  STRUCT
   STAT0 : ARRAY  [-32768 .. -30271 ] OF BYTE ;
  END_STRUCT ;
BEGIN
   STAT0[-32768] := B#16#0;
   STAT0[-32767] := B#16#0;
   STAT0[-32766] := B#16#0;
   STAT0[-32765] := B#16#0;
   STAT0[-32764] := B#16#0;
   STAT0[-32763] := B#16#1;
   STAT0[-32762] := B#16#0;
   STAT0[-32761] := B#16#0;
   STAT0[-32760] := B#16#0;
   STAT0[-32759] := B#16#1;
   STAT0[-32758] := B#16#0;
   STAT0[-32757] := B#16#1;
   STAT0[-32756] := B#16#0;
   STAT0[-32755] := B#16#1;
   STAT0[-32754] := B#16#0;
   STAT0[-32753] := B#16#1;
   STAT0[-32752] := B#16#0;
   STAT0[-32751] := B#16#1;
   STAT0[-32750] := B#16#0;
   STAT0[-32749] := B#16#1;
   STAT0[-32748] := B#16#0;
   STAT0[-32747] := B#16#1;
   STAT0[-32746] := B#16#0;
   STAT0[-32745] := B#16#1;
   STAT0[-32744] := B#16#0;
   STAT0[-32743] := B#16#1;
   STAT0[-32742] := B#16#0;
   STAT0[-32741] := B#16#1;
   STAT0[-32740] := B#16#0;
   STAT0[-32739] := B#16#1;
   STAT0[-32738] := B#16#0;
   STAT0[-32737] := B#16#0;
   STAT0[-32736] := B#16#0;
   STAT0[-32735] := B#16#0;
   STAT0[-32734] := B#16#0;
   STAT0[-32733] := B#16#0;
   STAT0[-32732] := B#16#0;
   STAT0[-32731] := B#16#0;
   STAT0[-32730] := B#16#0;
   STAT0[-32729] := B#16#0;
   STAT0[-32728] := B#16#0;
   STAT0[-32727] := B#16#0;
   STAT0[-32726] := B#16#0;
   STAT0[-32725] := B#16#0;
   STAT0[-32724] := B#16#0;
   STAT0[-32723] := B#16#0;
   STAT0[-32722] := B#16#0;
   STAT0[-32721] := B#16#0;
   STAT0[-32720] := B#16#0;
   STAT0[-32719] := B#16#0;
   STAT0[-32718] := B#16#0;
   STAT0[-32717] := B#16#0;
   STAT0[-32716] := B#16#0;
   STAT0[-32715] := B#16#0;
   STAT0[-32714] := B#16#0;
   STAT0[-32713] := B#16#0;
   STAT0[-32712] := B#16#0;
   STAT0[-32711] := B#16#0;
   STAT0[-32710] := B#16#0;
   STAT0[-32709] := B#16#0;
   STAT0[-32708] := B#16#0;
   STAT0[-32707] := B#16#0;
   STAT0[-32706] := B#16#0;
   STAT0[-32705] := B#16#0;
   STAT0[-32704] := B#16#0;
   STAT0[-32703] := B#16#0;
   STAT0[-32702] := B#16#0;
   STAT0[-32701] := B#16#0;
   STAT0[-32700] := B#16#0;
   STAT0[-32699] := B#16#0;
   STAT0[-32698] := B#16#0;
   STAT0[-32697] := B#16#0;
   STAT0[-32696] := B#16#0;
   STAT0[-32695] := B#16#0;
   STAT0[-32694] := B#16#0;
   STAT0[-32693] := B#16#0;
   STAT0[-32692] := B#16#0;
   STAT0[-32691] := B#16#0;
   STAT0[-32690] := B#16#0;
   STAT0[-32689] := B#16#0;
   STAT0[-32688] := B#16#0;
   STAT0[-32687] := B#16#0;
   STAT0[-32686] := B#16#0;
   STAT0[-32685] := B#16#0;
   STAT0[-32684] := B#16#0;
   STAT0[-32683] := B#16#0;
   STAT0[-32682] := B#16#0;
   STAT0[-32681] := B#16#0;
   STAT0[-32680] := B#16#0;
   STAT0[-32679] := B#16#0;
   STAT0[-32678] := B#16#0;
   STAT0[-32677] := B#16#0;
   STAT0[-32676] := B#16#0;
   STAT0[-32675] := B#16#0;
   STAT0[-32674] := B#16#0;
   STAT0[-32673] := B#16#0;
   STAT0[-32672] := B#16#0;
   STAT0[-32671] := B#16#0;
   STAT0[-32670] := B#16#0;
   STAT0[-32669] := B#16#0;
   STAT0[-32668] := B#16#0;
   STAT0[-32667] := B#16#0;
   STAT0[-32666] := B#16#0;
   STAT0[-32665] := B#16#0;
   STAT0[-32664] := B#16#0;
   STAT0[-32663] := B#16#0;
   STAT0[-32662] := B#16#0;
   STAT0[-32661] := B#16#0;
   STAT0[-32660] := B#16#0;
   STAT0[-32659] := B#16#0;
   STAT0[-32658] := B#16#0;
   STAT0[-32657] := B#16#0;
   STAT0[-32656] := B#16#0;
   STAT0[-32655] := B#16#0;
   STAT0[-32654] := B#16#0;
   STAT0[-32653] := B#16#0;
   STAT0[-32652] := B#16#0;
   STAT0[-32651] := B#16#0;
   STAT0[-32650] := B#16#0;
   STAT0[-32649] := B#16#0;
   STAT0[-32648] := B#16#0;
   STAT0[-32647] := B#16#0;
   STAT0[-32646] := B#16#0;
   STAT0[-32645] := B#16#0;
   STAT0[-32644] := B#16#0;
   STAT0[-32643] := B#16#0;
   STAT0[-32642] := B#16#0;
   STAT0[-32641] := B#16#0;
   STAT0[-32640] := B#16#0;
   STAT0[-32639] := B#16#0;
   STAT0[-32638] := B#16#0;
   STAT0[-32637] := B#16#0;
   STAT0[-32636] := B#16#0;
   STAT0[-32635] := B#16#0;
   STAT0[-32634] := B#16#0;
   STAT0[-32633] := B#16#0;
   STAT0[-32632] := B#16#0;
   STAT0[-32631] := B#16#0;
   STAT0[-32630] := B#16#0;
   STAT0[-32629] := B#16#0;
   STAT0[-32628] := B#16#0;
   STAT0[-32627] := B#16#0;
   STAT0[-32626] := B#16#0;
   STAT0[-32625] := B#16#0;
   STAT0[-32624] := B#16#0;
   STAT0[-32623] := B#16#0;
   STAT0[-32622] := B#16#0;
   STAT0[-32621] := B#16#0;
   STAT0[-32620] := B#16#0;
   STAT0[-32619] := B#16#0;
   STAT0[-32618] := B#16#0;
   STAT0[-32617] := B#16#0;
   STAT0[-32616] := B#16#0;
   STAT0[-32615] := B#16#0;
   STAT0[-32614] := B#16#0;
   STAT0[-32613] := B#16#0;
   STAT0[-32612] := B#16#0;
   STAT0[-32611] := B#16#0;
   STAT0[-32610] := B#16#0;
   STAT0[-32609] := B#16#0;
   STAT0[-32608] := B#16#0;
   STAT0[-32607] := B#16#0;
   STAT0[-32606] := B#16#0;
   STAT0[-32605] := B#16#0;
   STAT0[-32604] := B#16#0;
   STAT0[-32603] := B#16#0;
   STAT0[-32602] := B#16#0;
   STAT0[-32601] := B#16#0;
   STAT0[-32600] := B#16#0;
   STAT0[-32599] := B#16#0;
   STAT0[-32598] := B#16#0;
   STAT0[-32597] := B#16#0;
   STAT0[-32596] := B#16#0;
   STAT0[-32595] := B#16#0;
   STAT0[-32594] := B#16#0;
   STAT0[-32593] := B#16#0;
   STAT0[-32592] := B#16#0;
   STAT0[-32591] := B#16#0;
   STAT0[-32590] := B#16#0;
   STAT0[-32589] := B#16#0;
   STAT0[-32588] := B#16#0;
   STAT0[-32587] := B#16#0;
   STAT0[-32586] := B#16#0;
   STAT0[-32585] := B#16#0;
   STAT0[-32584] := B#16#0;
   STAT0[-32583] := B#16#0;
   STAT0[-32582] := B#16#0;
   STAT0[-32581] := B#16#0;
   STAT0[-32580] := B#16#0;
   STAT0[-32579] := B#16#0;
   STAT0[-32578] := B#16#0;
   STAT0[-32577] := B#16#0;
   STAT0[-32576] := B#16#0;
   STAT0[-32575] := B#16#0;
   STAT0[-32574] := B#16#0;
   STAT0[-32573] := B#16#0;
   STAT0[-32572] := B#16#0;
   STAT0[-32571] := B#16#0;
   STAT0[-32570] := B#16#0;
   STAT0[-32569] := B#16#0;
   STAT0[-32568] := B#16#0;
   STAT0[-32567] := B#16#0;
   STAT0[-32566] := B#16#0;
   STAT0[-32565] := B#16#0;
   STAT0[-32564] := B#16#0;
   STAT0[-32563] := B#16#0;
   STAT0[-32562] := B#16#0;
   STAT0[-32561] := B#16#0;
   STAT0[-32560] := B#16#0;
   STAT0[-32559] := B#16#0;
   STAT0[-32558] := B#16#0;
   STAT0[-32557] := B#16#0;
   STAT0[-32556] := B#16#0;
   STAT0[-32555] := B#16#0;
   STAT0[-32554] := B#16#0;
   STAT0[-32553] := B#16#0;
   STAT0[-32552] := B#16#0;
   STAT0[-32551] := B#16#0;
   STAT0[-32550] := B#16#0;
   STAT0[-32549] := B#16#0;
   STAT0[-32548] := B#16#0;
   STAT0[-32547] := B#16#0;
   STAT0[-32546] := B#16#0;
   STAT0[-32545] := B#16#0;
   STAT0[-32544] := B#16#0;
   STAT0[-32543] := B#16#0;
   STAT0[-32542] := B#16#0;
   STAT0[-32541] := B#16#0;
   STAT0[-32540] := B#16#0;
   STAT0[-32539] := B#16#0;
   STAT0[-32538] := B#16#0;
   STAT0[-32537] := B#16#0;
   STAT0[-32536] := B#16#0;
   STAT0[-32535] := B#16#0;
   STAT0[-32534] := B#16#0;
   STAT0[-32533] := B#16#0;
   STAT0[-32532] := B#16#0;
   STAT0[-32531] := B#16#0;
   STAT0[-32530] := B#16#0;
   STAT0[-32529] := B#16#0;
   STAT0[-32528] := B#16#0;
   STAT0[-32527] := B#16#0;
   STAT0[-32526] := B#16#0;
   STAT0[-32525] := B#16#0;
   STAT0[-32524] := B#16#0;
   STAT0[-32523] := B#16#0;
   STAT0[-32522] := B#16#0;
   STAT0[-32521] := B#16#0;
   STAT0[-32520] := B#16#0;
   STAT0[-32519] := B#16#0;
   STAT0[-32518] := B#16#0;
   STAT0[-32517] := B#16#0;
   STAT0[-32516] := B#16#0;
   STAT0[-32515] := B#16#0;
   STAT0[-32514] := B#16#0;
   STAT0[-32513] := B#16#0;
   STAT0[-32512] := B#16#0;
   STAT0[-32511] := B#16#0;
   STAT0[-32510] := B#16#0;
   STAT0[-32509] := B#16#0;
   STAT0[-32508] := B#16#0;
   STAT0[-32507] := B#16#0;
   STAT0[-32506] := B#16#0;
   STAT0[-32505] := B#16#0;
   STAT0[-32504] := B#16#0;
   STAT0[-32503] := B#16#0;
   STAT0[-32502] := B#16#0;
   STAT0[-32501] := B#16#0;
   STAT0[-32500] := B#16#0;
   STAT0[-32499] := B#16#0;
   STAT0[-32498] := B#16#0;
   STAT0[-32497] := B#16#0;
   STAT0[-32496] := B#16#0;
   STAT0[-32495] := B#16#0;
   STAT0[-32494] := B#16#0;
   STAT0[-32493] := B#16#0;
   STAT0[-32492] := B#16#0;
   STAT0[-32491] := B#16#0;
   STAT0[-32490] := B#16#0;
   STAT0[-32489] := B#16#0;
   STAT0[-32488] := B#16#0;
   STAT0[-32487] := B#16#0;
   STAT0[-32486] := B#16#0;
   STAT0[-32485] := B#16#0;
   STAT0[-32484] := B#16#0;
   STAT0[-32483] := B#16#0;
   STAT0[-32482] := B#16#0;
   STAT0[-32481] := B#16#0;
   STAT0[-32480] := B#16#0;
   STAT0[-32479] := B#16#0;
   STAT0[-32478] := B#16#0;
   STAT0[-32477] := B#16#0;
   STAT0[-32476] := B#16#0;
   STAT0[-32475] := B#16#0;
   STAT0[-32474] := B#16#0;
   STAT0[-32473] := B#16#0;
   STAT0[-32472] := B#16#0;
   STAT0[-32471] := B#16#0;
   STAT0[-32470] := B#16#0;
   STAT0[-32469] := B#16#0;
   STAT0[-32468] := B#16#0;
   STAT0[-32467] := B#16#0;
   STAT0[-32466] := B#16#0;
   STAT0[-32465] := B#16#0;
   STAT0[-32464] := B#16#0;
   STAT0[-32463] := B#16#0;
   STAT0[-32462] := B#16#0;
   STAT0[-32461] := B#16#0;
   STAT0[-32460] := B#16#0;
   STAT0[-32459] := B#16#0;
   STAT0[-32458] := B#16#0;
   STAT0[-32457] := B#16#0;
   STAT0[-32456] := B#16#0;
   STAT0[-32455] := B#16#0;
   STAT0[-32454] := B#16#0;
   STAT0[-32453] := B#16#0;
   STAT0[-32452] := B#16#0;
   STAT0[-32451] := B#16#0;
   STAT0[-32450] := B#16#0;
   STAT0[-32449] := B#16#0;
   STAT0[-32448] := B#16#0;
   STAT0[-32447] := B#16#0;
   STAT0[-32446] := B#16#0;
   STAT0[-32445] := B#16#0;
   STAT0[-32444] := B#16#0;
   STAT0[-32443] := B#16#0;
   STAT0[-32442] := B#16#0;
   STAT0[-32441] := B#16#0;
   STAT0[-32440] := B#16#0;
   STAT0[-32439] := B#16#0;
   STAT0[-32438] := B#16#0;
   STAT0[-32437] := B#16#0;
   STAT0[-32436] := B#16#0;
   STAT0[-32435] := B#16#0;
   STAT0[-32434] := B#16#0;
   STAT0[-32433] := B#16#0;
   STAT0[-32432] := B#16#0;
   STAT0[-32431] := B#16#0;
   STAT0[-32430] := B#16#0;
   STAT0[-32429] := B#16#0;
   STAT0[-32428] := B#16#0;
   STAT0[-32427] := B#16#0;
   STAT0[-32426] := B#16#0;
   STAT0[-32425] := B#16#0;
   STAT0[-32424] := B#16#0;
   STAT0[-32423] := B#16#0;
   STAT0[-32422] := B#16#0;
   STAT0[-32421] := B#16#0;
   STAT0[-32420] := B#16#0;
   STAT0[-32419] := B#16#0;
   STAT0[-32418] := B#16#0;
   STAT0[-32417] := B#16#0;
   STAT0[-32416] := B#16#0;
   STAT0[-32415] := B#16#0;
   STAT0[-32414] := B#16#0;
   STAT0[-32413] := B#16#0;
   STAT0[-32412] := B#16#0;
   STAT0[-32411] := B#16#0;
   STAT0[-32410] := B#16#0;
   STAT0[-32409] := B#16#0;
   STAT0[-32408] := B#16#0;
   STAT0[-32407] := B#16#0;
   STAT0[-32406] := B#16#0;
   STAT0[-32405] := B#16#0;
   STAT0[-32404] := B#16#0;
   STAT0[-32403] := B#16#0;
   STAT0[-32402] := B#16#0;
   STAT0[-32401] := B#16#0;
   STAT0[-32400] := B#16#0;
   STAT0[-32399] := B#16#0;
   STAT0[-32398] := B#16#0;
   STAT0[-32397] := B#16#0;
   STAT0[-32396] := B#16#0;
   STAT0[-32395] := B#16#0;
   STAT0[-32394] := B#16#0;
   STAT0[-32393] := B#16#0;
   STAT0[-32392] := B#16#0;
   STAT0[-32391] := B#16#0;
   STAT0[-32390] := B#16#0;
   STAT0[-32389] := B#16#0;
   STAT0[-32388] := B#16#0;
   STAT0[-32387] := B#16#0;
   STAT0[-32386] := B#16#0;
   STAT0[-32385] := B#16#0;
   STAT0[-32384] := B#16#0;
   STAT0[-32383] := B#16#0;
   STAT0[-32382] := B#16#0;
   STAT0[-32381] := B#16#0;
   STAT0[-32380] := B#16#0;
   STAT0[-32379] := B#16#0;
   STAT0[-32378] := B#16#0;
   STAT0[-32377] := B#16#0;
   STAT0[-32376] := B#16#0;
   STAT0[-32375] := B#16#0;
   STAT0[-32374] := B#16#0;
   STAT0[-32373] := B#16#0;
   STAT0[-32372] := B#16#0;
   STAT0[-32371] := B#16#0;
   STAT0[-32370] := B#16#0;
   STAT0[-32369] := B#16#0;
   STAT0[-32368] := B#16#0;
   STAT0[-32367] := B#16#0;
   STAT0[-32366] := B#16#0;
   STAT0[-32365] := B#16#0;
   STAT0[-32364] := B#16#0;
   STAT0[-32363] := B#16#0;
   STAT0[-32362] := B#16#0;
   STAT0[-32361] := B#16#0;
   STAT0[-32360] := B#16#0;
   STAT0[-32359] := B#16#0;
   STAT0[-32358] := B#16#0;
   STAT0[-32357] := B#16#0;
   STAT0[-32356] := B#16#0;
   STAT0[-32355] := B#16#0;
   STAT0[-32354] := B#16#0;
   STAT0[-32353] := B#16#0;
   STAT0[-32352] := B#16#0;
   STAT0[-32351] := B#16#0;
   STAT0[-32350] := B#16#0;
   STAT0[-32349] := B#16#0;
   STAT0[-32348] := B#16#0;
   STAT0[-32347] := B#16#0;
   STAT0[-32346] := B#16#0;
   STAT0[-32345] := B#16#0;
   STAT0[-32344] := B#16#0;
   STAT0[-32343] := B#16#0;
   STAT0[-32342] := B#16#0;
   STAT0[-32341] := B#16#0;
   STAT0[-32340] := B#16#0;
   STAT0[-32339] := B#16#0;
   STAT0[-32338] := B#16#0;
   STAT0[-32337] := B#16#0;
   STAT0[-32336] := B#16#0;
   STAT0[-32335] := B#16#0;
   STAT0[-32334] := B#16#0;
   STAT0[-32333] := B#16#0;
   STAT0[-32332] := B#16#0;
   STAT0[-32331] := B#16#0;
   STAT0[-32330] := B#16#0;
   STAT0[-32329] := B#16#0;
   STAT0[-32328] := B#16#0;
   STAT0[-32327] := B#16#0;
   STAT0[-32326] := B#16#0;
   STAT0[-32325] := B#16#0;
   STAT0[-32324] := B#16#0;
   STAT0[-32323] := B#16#0;
   STAT0[-32322] := B#16#0;
   STAT0[-32321] := B#16#0;
   STAT0[-32320] := B#16#0;
   STAT0[-32319] := B#16#0;
   STAT0[-32318] := B#16#0;
   STAT0[-32317] := B#16#0;
   STAT0[-32316] := B#16#0;
   STAT0[-32315] := B#16#0;
   STAT0[-32314] := B#16#0;
   STAT0[-32313] := B#16#0;
   STAT0[-32312] := B#16#0;
   STAT0[-32311] := B#16#0;
   STAT0[-32310] := B#16#0;
   STAT0[-32309] := B#16#0;
   STAT0[-32308] := B#16#0;
   STAT0[-32307] := B#16#0;
   STAT0[-32306] := B#16#0;
   STAT0[-32305] := B#16#0;
   STAT0[-32304] := B#16#0;
   STAT0[-32303] := B#16#0;
   STAT0[-32302] := B#16#0;
   STAT0[-32301] := B#16#0;
   STAT0[-32300] := B#16#0;
   STAT0[-32299] := B#16#0;
   STAT0[-32298] := B#16#0;
   STAT0[-32297] := B#16#0;
   STAT0[-32296] := B#16#0;
   STAT0[-32295] := B#16#0;
   STAT0[-32294] := B#16#0;
   STAT0[-32293] := B#16#0;
   STAT0[-32292] := B#16#0;
   STAT0[-32291] := B#16#0;
   STAT0[-32290] := B#16#0;
   STAT0[-32289] := B#16#0;
   STAT0[-32288] := B#16#0;
   STAT0[-32287] := B#16#0;
   STAT0[-32286] := B#16#0;
   STAT0[-32285] := B#16#0;
   STAT0[-32284] := B#16#0;
   STAT0[-32283] := B#16#0;
   STAT0[-32282] := B#16#0;
   STAT0[-32281] := B#16#0;
   STAT0[-32280] := B#16#0;
   STAT0[-32279] := B#16#0;
   STAT0[-32278] := B#16#0;
   STAT0[-32277] := B#16#0;
   STAT0[-32276] := B#16#0;
   STAT0[-32275] := B#16#0;
   STAT0[-32274] := B#16#0;
   STAT0[-32273] := B#16#0;
   STAT0[-32272] := B#16#0;
   STAT0[-32271] := B#16#0;
   STAT0[-32270] := B#16#0;
   STAT0[-32269] := B#16#0;
   STAT0[-32268] := B#16#0;
   STAT0[-32267] := B#16#0;
   STAT0[-32266] := B#16#0;
   STAT0[-32265] := B#16#0;
   STAT0[-32264] := B#16#0;
   STAT0[-32263] := B#16#0;
   STAT0[-32262] := B#16#0;
   STAT0[-32261] := B#16#0;
   STAT0[-32260] := B#16#0;
   STAT0[-32259] := B#16#0;
   STAT0[-32258] := B#16#0;
   STAT0[-32257] := B#16#0;
   STAT0[-32256] := B#16#0;
   STAT0[-32255] := B#16#0;
   STAT0[-32254] := B#16#0;
   STAT0[-32253] := B#16#0;
   STAT0[-32252] := B#16#0;
   STAT0[-32251] := B#16#0;
   STAT0[-32250] := B#16#0;
   STAT0[-32249] := B#16#0;
   STAT0[-32248] := B#16#0;
   STAT0[-32247] := B#16#0;
   STAT0[-32246] := B#16#0;
   STAT0[-32245] := B#16#0;
   STAT0[-32244] := B#16#0;
   STAT0[-32243] := B#16#0;
   STAT0[-32242] := B#16#0;
   STAT0[-32241] := B#16#0;
   STAT0[-32240] := B#16#0;
   STAT0[-32239] := B#16#0;
   STAT0[-32238] := B#16#0;
   STAT0[-32237] := B#16#0;
   STAT0[-32236] := B#16#0;
   STAT0[-32235] := B#16#0;
   STAT0[-32234] := B#16#0;
   STAT0[-32233] := B#16#0;
   STAT0[-32232] := B#16#0;
   STAT0[-32231] := B#16#0;
   STAT0[-32230] := B#16#0;
   STAT0[-32229] := B#16#0;
   STAT0[-32228] := B#16#0;
   STAT0[-32227] := B#16#0;
   STAT0[-32226] := B#16#0;
   STAT0[-32225] := B#16#0;
   STAT0[-32224] := B#16#0;
   STAT0[-32223] := B#16#0;
   STAT0[-32222] := B#16#0;
   STAT0[-32221] := B#16#0;
   STAT0[-32220] := B#16#0;
   STAT0[-32219] := B#16#0;
   STAT0[-32218] := B#16#0;
   STAT0[-32217] := B#16#0;
   STAT0[-32216] := B#16#0;
   STAT0[-32215] := B#16#0;
   STAT0[-32214] := B#16#0;
   STAT0[-32213] := B#16#0;
   STAT0[-32212] := B#16#0;
   STAT0[-32211] := B#16#0;
   STAT0[-32210] := B#16#0;
   STAT0[-32209] := B#16#0;
   STAT0[-32208] := B#16#0;
   STAT0[-32207] := B#16#0;
   STAT0[-32206] := B#16#0;
   STAT0[-32205] := B#16#0;
   STAT0[-32204] := B#16#0;
   STAT0[-32203] := B#16#0;
   STAT0[-32202] := B#16#0;
   STAT0[-32201] := B#16#0;
   STAT0[-32200] := B#16#0;
   STAT0[-32199] := B#16#0;
   STAT0[-32198] := B#16#0;
   STAT0[-32197] := B#16#0;
   STAT0[-32196] := B#16#0;
   STAT0[-32195] := B#16#0;
   STAT0[-32194] := B#16#0;
   STAT0[-32193] := B#16#0;
   STAT0[-32192] := B#16#0;
   STAT0[-32191] := B#16#0;
   STAT0[-32190] := B#16#0;
   STAT0[-32189] := B#16#0;
   STAT0[-32188] := B#16#0;
   STAT0[-32187] := B#16#0;
   STAT0[-32186] := B#16#0;
   STAT0[-32185] := B#16#0;
   STAT0[-32184] := B#16#0;
   STAT0[-32183] := B#16#0;
   STAT0[-32182] := B#16#0;
   STAT0[-32181] := B#16#0;
   STAT0[-32180] := B#16#0;
   STAT0[-32179] := B#16#0;
   STAT0[-32178] := B#16#0;
   STAT0[-32177] := B#16#0;
   STAT0[-32176] := B#16#0;
   STAT0[-32175] := B#16#0;
   STAT0[-32174] := B#16#0;
   STAT0[-32173] := B#16#0;
   STAT0[-32172] := B#16#0;
   STAT0[-32171] := B#16#0;
   STAT0[-32170] := B#16#0;
   STAT0[-32169] := B#16#0;
   STAT0[-32168] := B#16#0;
   STAT0[-32167] := B#16#0;
   STAT0[-32166] := B#16#0;
   STAT0[-32165] := B#16#0;
   STAT0[-32164] := B#16#0;
   STAT0[-32163] := B#16#0;
   STAT0[-32162] := B#16#0;
   STAT0[-32161] := B#16#0;
   STAT0[-32160] := B#16#0;
   STAT0[-32159] := B#16#0;
   STAT0[-32158] := B#16#0;
   STAT0[-32157] := B#16#0;
   STAT0[-32156] := B#16#0;
   STAT0[-32155] := B#16#0;
   STAT0[-32154] := B#16#0;
   STAT0[-32153] := B#16#0;
   STAT0[-32152] := B#16#0;
   STAT0[-32151] := B#16#0;
   STAT0[-32150] := B#16#0;
   STAT0[-32149] := B#16#0;
   STAT0[-32148] := B#16#0;
   STAT0[-32147] := B#16#0;
   STAT0[-32146] := B#16#0;
   STAT0[-32145] := B#16#0;
   STAT0[-32144] := B#16#0;
   STAT0[-32143] := B#16#0;
   STAT0[-32142] := B#16#0;
   STAT0[-32141] := B#16#0;
   STAT0[-32140] := B#16#0;
   STAT0[-32139] := B#16#0;
   STAT0[-32138] := B#16#0;
   STAT0[-32137] := B#16#0;
   STAT0[-32136] := B#16#0;
   STAT0[-32135] := B#16#0;
   STAT0[-32134] := B#16#0;
   STAT0[-32133] := B#16#0;
   STAT0[-32132] := B#16#0;
   STAT0[-32131] := B#16#0;
   STAT0[-32130] := B#16#0;
   STAT0[-32129] := B#16#0;
   STAT0[-32128] := B#16#0;
   STAT0[-32127] := B#16#0;
   STAT0[-32126] := B#16#0;
   STAT0[-32125] := B#16#0;
   STAT0[-32124] := B#16#0;
   STAT0[-32123] := B#16#0;
   STAT0[-32122] := B#16#0;
   STAT0[-32121] := B#16#0;
   STAT0[-32120] := B#16#0;
   STAT0[-32119] := B#16#0;
   STAT0[-32118] := B#16#0;
   STAT0[-32117] := B#16#0;
   STAT0[-32116] := B#16#0;
   STAT0[-32115] := B#16#0;
   STAT0[-32114] := B#16#0;
   STAT0[-32113] := B#16#0;
   STAT0[-32112] := B#16#0;
   STAT0[-32111] := B#16#0;
   STAT0[-32110] := B#16#0;
   STAT0[-32109] := B#16#0;
   STAT0[-32108] := B#16#0;
   STAT0[-32107] := B#16#0;
   STAT0[-32106] := B#16#0;
   STAT0[-32105] := B#16#0;
   STAT0[-32104] := B#16#0;
   STAT0[-32103] := B#16#0;
   STAT0[-32102] := B#16#0;
   STAT0[-32101] := B#16#0;
   STAT0[-32100] := B#16#0;
   STAT0[-32099] := B#16#0;
   STAT0[-32098] := B#16#0;
   STAT0[-32097] := B#16#0;
   STAT0[-32096] := B#16#0;
   STAT0[-32095] := B#16#0;
   STAT0[-32094] := B#16#0;
   STAT0[-32093] := B#16#0;
   STAT0[-32092] := B#16#0;
   STAT0[-32091] := B#16#0;
   STAT0[-32090] := B#16#0;
   STAT0[-32089] := B#16#0;
   STAT0[-32088] := B#16#0;
   STAT0[-32087] := B#16#0;
   STAT0[-32086] := B#16#0;
   STAT0[-32085] := B#16#0;
   STAT0[-32084] := B#16#0;
   STAT0[-32083] := B#16#0;
   STAT0[-32082] := B#16#0;
   STAT0[-32081] := B#16#0;
   STAT0[-32080] := B#16#0;
   STAT0[-32079] := B#16#0;
   STAT0[-32078] := B#16#0;
   STAT0[-32077] := B#16#0;
   STAT0[-32076] := B#16#0;
   STAT0[-32075] := B#16#0;
   STAT0[-32074] := B#16#0;
   STAT0[-32073] := B#16#0;
   STAT0[-32072] := B#16#0;
   STAT0[-32071] := B#16#0;
   STAT0[-32070] := B#16#0;
   STAT0[-32069] := B#16#0;
   STAT0[-32068] := B#16#0;
   STAT0[-32067] := B#16#0;
   STAT0[-32066] := B#16#0;
   STAT0[-32065] := B#16#0;
   STAT0[-32064] := B#16#0;
   STAT0[-32063] := B#16#0;
   STAT0[-32062] := B#16#0;
   STAT0[-32061] := B#16#0;
   STAT0[-32060] := B#16#0;
   STAT0[-32059] := B#16#0;
   STAT0[-32058] := B#16#0;
   STAT0[-32057] := B#16#0;
   STAT0[-32056] := B#16#0;
   STAT0[-32055] := B#16#0;
   STAT0[-32054] := B#16#0;
   STAT0[-32053] := B#16#0;
   STAT0[-32052] := B#16#0;
   STAT0[-32051] := B#16#0;
   STAT0[-32050] := B#16#0;
   STAT0[-32049] := B#16#0;
   STAT0[-32048] := B#16#0;
   STAT0[-32047] := B#16#0;
   STAT0[-32046] := B#16#0;
   STAT0[-32045] := B#16#0;
   STAT0[-32044] := B#16#0;
   STAT0[-32043] := B#16#0;
   STAT0[-32042] := B#16#0;
   STAT0[-32041] := B#16#0;
   STAT0[-32040] := B#16#0;
   STAT0[-32039] := B#16#0;
   STAT0[-32038] := B#16#0;
   STAT0[-32037] := B#16#0;
   STAT0[-32036] := B#16#0;
   STAT0[-32035] := B#16#0;
   STAT0[-32034] := B#16#0;
   STAT0[-32033] := B#16#0;
   STAT0[-32032] := B#16#0;
   STAT0[-32031] := B#16#0;
   STAT0[-32030] := B#16#0;
   STAT0[-32029] := B#16#0;
   STAT0[-32028] := B#16#0;
   STAT0[-32027] := B#16#0;
   STAT0[-32026] := B#16#0;
   STAT0[-32025] := B#16#0;
   STAT0[-32024] := B#16#0;
   STAT0[-32023] := B#16#0;
   STAT0[-32022] := B#16#0;
   STAT0[-32021] := B#16#0;
   STAT0[-32020] := B#16#0;
   STAT0[-32019] := B#16#0;
   STAT0[-32018] := B#16#0;
   STAT0[-32017] := B#16#0;
   STAT0[-32016] := B#16#0;
   STAT0[-32015] := B#16#0;
   STAT0[-32014] := B#16#0;
   STAT0[-32013] := B#16#0;
   STAT0[-32012] := B#16#0;
   STAT0[-32011] := B#16#0;
   STAT0[-32010] := B#16#0;
   STAT0[-32009] := B#16#0;
   STAT0[-32008] := B#16#0;
   STAT0[-32007] := B#16#0;
   STAT0[-32006] := B#16#0;
   STAT0[-32005] := B#16#0;
   STAT0[-32004] := B#16#0;
   STAT0[-32003] := B#16#0;
   STAT0[-32002] := B#16#0;
   STAT0[-32001] := B#16#0;
   STAT0[-32000] := B#16#0;
   STAT0[-31999] := B#16#0;
   STAT0[-31998] := B#16#0;
   STAT0[-31997] := B#16#0;
   STAT0[-31996] := B#16#0;
   STAT0[-31995] := B#16#0;
   STAT0[-31994] := B#16#0;
   STAT0[-31993] := B#16#0;
   STAT0[-31992] := B#16#0;
   STAT0[-31991] := B#16#0;
   STAT0[-31990] := B#16#0;
   STAT0[-31989] := B#16#0;
   STAT0[-31988] := B#16#0;
   STAT0[-31987] := B#16#0;
   STAT0[-31986] := B#16#0;
   STAT0[-31985] := B#16#0;
   STAT0[-31984] := B#16#0;
   STAT0[-31983] := B#16#0;
   STAT0[-31982] := B#16#0;
   STAT0[-31981] := B#16#0;
   STAT0[-31980] := B#16#0;
   STAT0[-31979] := B#16#0;
   STAT0[-31978] := B#16#0;
   STAT0[-31977] := B#16#0;
   STAT0[-31976] := B#16#0;
   STAT0[-31975] := B#16#0;
   STAT0[-31974] := B#16#0;
   STAT0[-31973] := B#16#0;
   STAT0[-31972] := B#16#0;
   STAT0[-31971] := B#16#0;
   STAT0[-31970] := B#16#0;
   STAT0[-31969] := B#16#0;
   STAT0[-31968] := B#16#0;
   STAT0[-31967] := B#16#0;
   STAT0[-31966] := B#16#0;
   STAT0[-31965] := B#16#0;
   STAT0[-31964] := B#16#0;
   STAT0[-31963] := B#16#0;
   STAT0[-31962] := B#16#0;
   STAT0[-31961] := B#16#0;
   STAT0[-31960] := B#16#0;
   STAT0[-31959] := B#16#0;
   STAT0[-31958] := B#16#0;
   STAT0[-31957] := B#16#0;
   STAT0[-31956] := B#16#0;
   STAT0[-31955] := B#16#0;
   STAT0[-31954] := B#16#0;
   STAT0[-31953] := B#16#0;
   STAT0[-31952] := B#16#0;
   STAT0[-31951] := B#16#0;
   STAT0[-31950] := B#16#0;
   STAT0[-31949] := B#16#0;
   STAT0[-31948] := B#16#0;
   STAT0[-31947] := B#16#0;
   STAT0[-31946] := B#16#0;
   STAT0[-31945] := B#16#0;
   STAT0[-31944] := B#16#0;
   STAT0[-31943] := B#16#0;
   STAT0[-31942] := B#16#0;
   STAT0[-31941] := B#16#0;
   STAT0[-31940] := B#16#0;
   STAT0[-31939] := B#16#0;
   STAT0[-31938] := B#16#0;
   STAT0[-31937] := B#16#0;
   STAT0[-31936] := B#16#0;
   STAT0[-31935] := B#16#0;
   STAT0[-31934] := B#16#0;
   STAT0[-31933] := B#16#0;
   STAT0[-31932] := B#16#0;
   STAT0[-31931] := B#16#0;
   STAT0[-31930] := B#16#0;
   STAT0[-31929] := B#16#0;
   STAT0[-31928] := B#16#0;
   STAT0[-31927] := B#16#0;
   STAT0[-31926] := B#16#0;
   STAT0[-31925] := B#16#0;
   STAT0[-31924] := B#16#0;
   STAT0[-31923] := B#16#0;
   STAT0[-31922] := B#16#0;
   STAT0[-31921] := B#16#0;
   STAT0[-31920] := B#16#0;
   STAT0[-31919] := B#16#0;
   STAT0[-31918] := B#16#0;
   STAT0[-31917] := B#16#0;
   STAT0[-31916] := B#16#0;
   STAT0[-31915] := B#16#0;
   STAT0[-31914] := B#16#0;
   STAT0[-31913] := B#16#0;
   STAT0[-31912] := B#16#0;
   STAT0[-31911] := B#16#0;
   STAT0[-31910] := B#16#0;
   STAT0[-31909] := B#16#0;
   STAT0[-31908] := B#16#0;
   STAT0[-31907] := B#16#0;
   STAT0[-31906] := B#16#0;
   STAT0[-31905] := B#16#0;
   STAT0[-31904] := B#16#0;
   STAT0[-31903] := B#16#0;
   STAT0[-31902] := B#16#0;
   STAT0[-31901] := B#16#0;
   STAT0[-31900] := B#16#0;
   STAT0[-31899] := B#16#0;
   STAT0[-31898] := B#16#0;
   STAT0[-31897] := B#16#0;
   STAT0[-31896] := B#16#0;
   STAT0[-31895] := B#16#0;
   STAT0[-31894] := B#16#0;
   STAT0[-31893] := B#16#0;
   STAT0[-31892] := B#16#0;
   STAT0[-31891] := B#16#0;
   STAT0[-31890] := B#16#0;
   STAT0[-31889] := B#16#0;
   STAT0[-31888] := B#16#0;
   STAT0[-31887] := B#16#0;
   STAT0[-31886] := B#16#0;
   STAT0[-31885] := B#16#0;
   STAT0[-31884] := B#16#0;
   STAT0[-31883] := B#16#0;
   STAT0[-31882] := B#16#0;
   STAT0[-31881] := B#16#0;
   STAT0[-31880] := B#16#0;
   STAT0[-31879] := B#16#0;
   STAT0[-31878] := B#16#0;
   STAT0[-31877] := B#16#0;
   STAT0[-31876] := B#16#0;
   STAT0[-31875] := B#16#0;
   STAT0[-31874] := B#16#0;
   STAT0[-31873] := B#16#0;
   STAT0[-31872] := B#16#0;
   STAT0[-31871] := B#16#0;
   STAT0[-31870] := B#16#0;
   STAT0[-31869] := B#16#0;
   STAT0[-31868] := B#16#0;
   STAT0[-31867] := B#16#0;
   STAT0[-31866] := B#16#0;
   STAT0[-31865] := B#16#0;
   STAT0[-31864] := B#16#0;
   STAT0[-31863] := B#16#0;
   STAT0[-31862] := B#16#0;
   STAT0[-31861] := B#16#0;
   STAT0[-31860] := B#16#0;
   STAT0[-31859] := B#16#0;
   STAT0[-31858] := B#16#0;
   STAT0[-31857] := B#16#0;
   STAT0[-31856] := B#16#0;
   STAT0[-31855] := B#16#0;
   STAT0[-31854] := B#16#0;
   STAT0[-31853] := B#16#0;
   STAT0[-31852] := B#16#0;
   STAT0[-31851] := B#16#0;
   STAT0[-31850] := B#16#0;
   STAT0[-31849] := B#16#0;
   STAT0[-31848] := B#16#0;
   STAT0[-31847] := B#16#0;
   STAT0[-31846] := B#16#0;
   STAT0[-31845] := B#16#0;
   STAT0[-31844] := B#16#0;
   STAT0[-31843] := B#16#0;
   STAT0[-31842] := B#16#0;
   STAT0[-31841] := B#16#0;
   STAT0[-31840] := B#16#0;
   STAT0[-31839] := B#16#0;
   STAT0[-31838] := B#16#0;
   STAT0[-31837] := B#16#0;
   STAT0[-31836] := B#16#0;
   STAT0[-31835] := B#16#0;
   STAT0[-31834] := B#16#0;
   STAT0[-31833] := B#16#0;
   STAT0[-31832] := B#16#0;
   STAT0[-31831] := B#16#0;
   STAT0[-31830] := B#16#0;
   STAT0[-31829] := B#16#0;
   STAT0[-31828] := B#16#0;
   STAT0[-31827] := B#16#0;
   STAT0[-31826] := B#16#0;
   STAT0[-31825] := B#16#0;
   STAT0[-31824] := B#16#0;
   STAT0[-31823] := B#16#0;
   STAT0[-31822] := B#16#0;
   STAT0[-31821] := B#16#0;
   STAT0[-31820] := B#16#0;
   STAT0[-31819] := B#16#0;
   STAT0[-31818] := B#16#0;
   STAT0[-31817] := B#16#0;
   STAT0[-31816] := B#16#0;
   STAT0[-31815] := B#16#0;
   STAT0[-31814] := B#16#0;
   STAT0[-31813] := B#16#0;
   STAT0[-31812] := B#16#0;
   STAT0[-31811] := B#16#0;
   STAT0[-31810] := B#16#0;
   STAT0[-31809] := B#16#0;
   STAT0[-31808] := B#16#0;
   STAT0[-31807] := B#16#0;
   STAT0[-31806] := B#16#0;
   STAT0[-31805] := B#16#0;
   STAT0[-31804] := B#16#0;
   STAT0[-31803] := B#16#0;
   STAT0[-31802] := B#16#0;
   STAT0[-31801] := B#16#0;
   STAT0[-31800] := B#16#0;
   STAT0[-31799] := B#16#0;
   STAT0[-31798] := B#16#0;
   STAT0[-31797] := B#16#0;
   STAT0[-31796] := B#16#0;
   STAT0[-31795] := B#16#0;
   STAT0[-31794] := B#16#0;
   STAT0[-31793] := B#16#0;
   STAT0[-31792] := B#16#0;
   STAT0[-31791] := B#16#0;
   STAT0[-31790] := B#16#0;
   STAT0[-31789] := B#16#0;
   STAT0[-31788] := B#16#0;
   STAT0[-31787] := B#16#0;
   STAT0[-31786] := B#16#0;
   STAT0[-31785] := B#16#0;
   STAT0[-31784] := B#16#0;
   STAT0[-31783] := B#16#0;
   STAT0[-31782] := B#16#0;
   STAT0[-31781] := B#16#0;
   STAT0[-31780] := B#16#0;
   STAT0[-31779] := B#16#0;
   STAT0[-31778] := B#16#0;
   STAT0[-31777] := B#16#0;
   STAT0[-31776] := B#16#0;
   STAT0[-31775] := B#16#0;
   STAT0[-31774] := B#16#0;
   STAT0[-31773] := B#16#0;
   STAT0[-31772] := B#16#0;
   STAT0[-31771] := B#16#0;
   STAT0[-31770] := B#16#0;
   STAT0[-31769] := B#16#0;
   STAT0[-31768] := B#16#0;
   STAT0[-31767] := B#16#0;
   STAT0[-31766] := B#16#0;
   STAT0[-31765] := B#16#0;
   STAT0[-31764] := B#16#0;
   STAT0[-31763] := B#16#0;
   STAT0[-31762] := B#16#0;
   STAT0[-31761] := B#16#0;
   STAT0[-31760] := B#16#0;
   STAT0[-31759] := B#16#0;
   STAT0[-31758] := B#16#0;
   STAT0[-31757] := B#16#0;
   STAT0[-31756] := B#16#0;
   STAT0[-31755] := B#16#0;
   STAT0[-31754] := B#16#0;
   STAT0[-31753] := B#16#0;
   STAT0[-31752] := B#16#0;
   STAT0[-31751] := B#16#0;
   STAT0[-31750] := B#16#0;
   STAT0[-31749] := B#16#0;
   STAT0[-31748] := B#16#0;
   STAT0[-31747] := B#16#0;
   STAT0[-31746] := B#16#0;
   STAT0[-31745] := B#16#0;
   STAT0[-31744] := B#16#0;
   STAT0[-31743] := B#16#0;
   STAT0[-31742] := B#16#0;
   STAT0[-31741] := B#16#0;
   STAT0[-31740] := B#16#0;
   STAT0[-31739] := B#16#0;
   STAT0[-31738] := B#16#0;
   STAT0[-31737] := B#16#0;
   STAT0[-31736] := B#16#0;
   STAT0[-31735] := B#16#0;
   STAT0[-31734] := B#16#0;
   STAT0[-31733] := B#16#0;
   STAT0[-31732] := B#16#0;
   STAT0[-31731] := B#16#0;
   STAT0[-31730] := B#16#0;
   STAT0[-31729] := B#16#0;
   STAT0[-31728] := B#16#0;
   STAT0[-31727] := B#16#0;
   STAT0[-31726] := B#16#0;
   STAT0[-31725] := B#16#0;
   STAT0[-31724] := B#16#0;
   STAT0[-31723] := B#16#0;
   STAT0[-31722] := B#16#0;
   STAT0[-31721] := B#16#1;
   STAT0[-31720] := B#16#0;
   STAT0[-31719] := B#16#0;
   STAT0[-31718] := B#16#0;
   STAT0[-31717] := B#16#0;
   STAT0[-31716] := B#16#0;
   STAT0[-31715] := B#16#0;
   STAT0[-31714] := B#16#0;
   STAT0[-31713] := B#16#0;
   STAT0[-31712] := B#16#0;
   STAT0[-31711] := B#16#0;
   STAT0[-31710] := B#16#0;
   STAT0[-31709] := B#16#0;
   STAT0[-31708] := B#16#0;
   STAT0[-31707] := B#16#0;
   STAT0[-31706] := B#16#0;
   STAT0[-31705] := B#16#1;
   STAT0[-31704] := B#16#0;
   STAT0[-31703] := B#16#1;
   STAT0[-31702] := B#16#0;
   STAT0[-31701] := B#16#1;
   STAT0[-31700] := B#16#0;
   STAT0[-31699] := B#16#1;
   STAT0[-31698] := B#16#0;
   STAT0[-31697] := B#16#0;
   STAT0[-31696] := B#16#0;
   STAT0[-31695] := B#16#0;
   STAT0[-31694] := B#16#0;
   STAT0[-31693] := B#16#0;
   STAT0[-31692] := B#16#0;
   STAT0[-31691] := B#16#0;
   STAT0[-31690] := B#16#0;
   STAT0[-31689] := B#16#0;
   STAT0[-31688] := B#16#0;
   STAT0[-31687] := B#16#0;
   STAT0[-31686] := B#16#0;
   STAT0[-31685] := B#16#0;
   STAT0[-31684] := B#16#0;
   STAT0[-31683] := B#16#0;
   STAT0[-31682] := B#16#0;
   STAT0[-31681] := B#16#0;
   STAT0[-31680] := B#16#0;
   STAT0[-31679] := B#16#0;
   STAT0[-31678] := B#16#0;
   STAT0[-31677] := B#16#0;
   STAT0[-31676] := B#16#0;
   STAT0[-31675] := B#16#0;
   STAT0[-31674] := B#16#0;
   STAT0[-31673] := B#16#0;
   STAT0[-31672] := B#16#0;
   STAT0[-31671] := B#16#0;
   STAT0[-31670] := B#16#0;
   STAT0[-31669] := B#16#0;
   STAT0[-31668] := B#16#0;
   STAT0[-31667] := B#16#0;
   STAT0[-31666] := B#16#0;
   STAT0[-31665] := B#16#0;
   STAT0[-31664] := B#16#0;
   STAT0[-31663] := B#16#0;
   STAT0[-31662] := B#16#0;
   STAT0[-31661] := B#16#0;
   STAT0[-31660] := B#16#0;
   STAT0[-31659] := B#16#0;
   STAT0[-31658] := B#16#0;
   STAT0[-31657] := B#16#0;
   STAT0[-31656] := B#16#0;
   STAT0[-31655] := B#16#0;
   STAT0[-31654] := B#16#0;
   STAT0[-31653] := B#16#0;
   STAT0[-31652] := B#16#0;
   STAT0[-31651] := B#16#0;
   STAT0[-31650] := B#16#0;
   STAT0[-31649] := B#16#0;
   STAT0[-31648] := B#16#0;
   STAT0[-31647] := B#16#0;
   STAT0[-31646] := B#16#0;
   STAT0[-31645] := B#16#0;
   STAT0[-31644] := B#16#0;
   STAT0[-31643] := B#16#0;
   STAT0[-31642] := B#16#0;
   STAT0[-31641] := B#16#0;
   STAT0[-31640] := B#16#0;
   STAT0[-31639] := B#16#0;
   STAT0[-31638] := B#16#0;
   STAT0[-31637] := B#16#0;
   STAT0[-31636] := B#16#0;
   STAT0[-31635] := B#16#0;
   STAT0[-31634] := B#16#0;
   STAT0[-31633] := B#16#0;
   STAT0[-31632] := B#16#0;
   STAT0[-31631] := B#16#0;
   STAT0[-31630] := B#16#0;
   STAT0[-31629] := B#16#0;
   STAT0[-31628] := B#16#0;
   STAT0[-31627] := B#16#0;
   STAT0[-31626] := B#16#0;
   STAT0[-31625] := B#16#0;
   STAT0[-31624] := B#16#0;
   STAT0[-31623] := B#16#0;
   STAT0[-31622] := B#16#0;
   STAT0[-31621] := B#16#0;
   STAT0[-31620] := B#16#0;
   STAT0[-31619] := B#16#0;
   STAT0[-31618] := B#16#0;
   STAT0[-31617] := B#16#0;
   STAT0[-31616] := B#16#0;
   STAT0[-31615] := B#16#0;
   STAT0[-31614] := B#16#0;
   STAT0[-31613] := B#16#0;
   STAT0[-31612] := B#16#0;
   STAT0[-31611] := B#16#0;
   STAT0[-31610] := B#16#0;
   STAT0[-31609] := B#16#0;
   STAT0[-31608] := B#16#0;
   STAT0[-31607] := B#16#0;
   STAT0[-31606] := B#16#0;
   STAT0[-31605] := B#16#0;
   STAT0[-31604] := B#16#0;
   STAT0[-31603] := B#16#0;
   STAT0[-31602] := B#16#0;
   STAT0[-31601] := B#16#0;
   STAT0[-31600] := B#16#0;
   STAT0[-31599] := B#16#0;
   STAT0[-31598] := B#16#0;
   STAT0[-31597] := B#16#0;
   STAT0[-31596] := B#16#0;
   STAT0[-31595] := B#16#0;
   STAT0[-31594] := B#16#0;
   STAT0[-31593] := B#16#0;
   STAT0[-31592] := B#16#0;
   STAT0[-31591] := B#16#0;
   STAT0[-31590] := B#16#0;
   STAT0[-31589] := B#16#0;
   STAT0[-31588] := B#16#0;
   STAT0[-31587] := B#16#0;
   STAT0[-31586] := B#16#0;
   STAT0[-31585] := B#16#0;
   STAT0[-31584] := B#16#0;
   STAT0[-31583] := B#16#0;
   STAT0[-31582] := B#16#0;
   STAT0[-31581] := B#16#0;
   STAT0[-31580] := B#16#0;
   STAT0[-31579] := B#16#0;
   STAT0[-31578] := B#16#0;
   STAT0[-31577] := B#16#0;
   STAT0[-31576] := B#16#0;
   STAT0[-31575] := B#16#0;
   STAT0[-31574] := B#16#0;
   STAT0[-31573] := B#16#0;
   STAT0[-31572] := B#16#0;
   STAT0[-31571] := B#16#0;
   STAT0[-31570] := B#16#0;
   STAT0[-31569] := B#16#0;
   STAT0[-31568] := B#16#0;
   STAT0[-31567] := B#16#0;
   STAT0[-31566] := B#16#0;
   STAT0[-31565] := B#16#0;
   STAT0[-31564] := B#16#0;
   STAT0[-31563] := B#16#0;
   STAT0[-31562] := B#16#0;
   STAT0[-31561] := B#16#0;
   STAT0[-31560] := B#16#0;
   STAT0[-31559] := B#16#0;
   STAT0[-31558] := B#16#0;
   STAT0[-31557] := B#16#0;
   STAT0[-31556] := B#16#0;
   STAT0[-31555] := B#16#0;
   STAT0[-31554] := B#16#0;
   STAT0[-31553] := B#16#0;
   STAT0[-31552] := B#16#0;
   STAT0[-31551] := B#16#0;
   STAT0[-31550] := B#16#0;
   STAT0[-31549] := B#16#0;
   STAT0[-31548] := B#16#0;
   STAT0[-31547] := B#16#0;
   STAT0[-31546] := B#16#0;
   STAT0[-31545] := B#16#0;
   STAT0[-31544] := B#16#0;
   STAT0[-31543] := B#16#0;
   STAT0[-31542] := B#16#0;
   STAT0[-31541] := B#16#0;
   STAT0[-31540] := B#16#0;
   STAT0[-31539] := B#16#0;
   STAT0[-31538] := B#16#0;
   STAT0[-31537] := B#16#0;
   STAT0[-31536] := B#16#0;
   STAT0[-31535] := B#16#0;
   STAT0[-31534] := B#16#0;
   STAT0[-31533] := B#16#0;
   STAT0[-31532] := B#16#0;
   STAT0[-31531] := B#16#0;
   STAT0[-31530] := B#16#0;
   STAT0[-31529] := B#16#0;
   STAT0[-31528] := B#16#0;
   STAT0[-31527] := B#16#0;
   STAT0[-31526] := B#16#0;
   STAT0[-31525] := B#16#0;
   STAT0[-31524] := B#16#0;
   STAT0[-31523] := B#16#0;
   STAT0[-31522] := B#16#0;
   STAT0[-31521] := B#16#0;
   STAT0[-31520] := B#16#0;
   STAT0[-31519] := B#16#0;
   STAT0[-31518] := B#16#0;
   STAT0[-31517] := B#16#0;
   STAT0[-31516] := B#16#0;
   STAT0[-31515] := B#16#0;
   STAT0[-31514] := B#16#0;
   STAT0[-31513] := B#16#0;
   STAT0[-31512] := B#16#0;
   STAT0[-31511] := B#16#0;
   STAT0[-31510] := B#16#0;
   STAT0[-31509] := B#16#0;
   STAT0[-31508] := B#16#0;
   STAT0[-31507] := B#16#0;
   STAT0[-31506] := B#16#0;
   STAT0[-31505] := B#16#0;
   STAT0[-31504] := B#16#0;
   STAT0[-31503] := B#16#0;
   STAT0[-31502] := B#16#0;
   STAT0[-31501] := B#16#0;
   STAT0[-31500] := B#16#0;
   STAT0[-31499] := B#16#0;
   STAT0[-31498] := B#16#0;
   STAT0[-31497] := B#16#0;
   STAT0[-31496] := B#16#0;
   STAT0[-31495] := B#16#0;
   STAT0[-31494] := B#16#0;
   STAT0[-31493] := B#16#0;
   STAT0[-31492] := B#16#0;
   STAT0[-31491] := B#16#0;
   STAT0[-31490] := B#16#0;
   STAT0[-31489] := B#16#0;
   STAT0[-31488] := B#16#0;
   STAT0[-31487] := B#16#0;
   STAT0[-31486] := B#16#0;
   STAT0[-31485] := B#16#0;
   STAT0[-31484] := B#16#0;
   STAT0[-31483] := B#16#0;
   STAT0[-31482] := B#16#0;
   STAT0[-31481] := B#16#0;
   STAT0[-31480] := B#16#0;
   STAT0[-31479] := B#16#0;
   STAT0[-31478] := B#16#0;
   STAT0[-31477] := B#16#0;
   STAT0[-31476] := B#16#0;
   STAT0[-31475] := B#16#0;
   STAT0[-31474] := B#16#0;
   STAT0[-31473] := B#16#0;
   STAT0[-31472] := B#16#0;
   STAT0[-31471] := B#16#0;
   STAT0[-31470] := B#16#0;
   STAT0[-31469] := B#16#0;
   STAT0[-31468] := B#16#0;
   STAT0[-31467] := B#16#0;
   STAT0[-31466] := B#16#0;
   STAT0[-31465] := B#16#0;
   STAT0[-31464] := B#16#0;
   STAT0[-31463] := B#16#0;
   STAT0[-31462] := B#16#0;
   STAT0[-31461] := B#16#0;
   STAT0[-31460] := B#16#0;
   STAT0[-31459] := B#16#0;
   STAT0[-31458] := B#16#0;
   STAT0[-31457] := B#16#0;
   STAT0[-31456] := B#16#0;
   STAT0[-31455] := B#16#0;
   STAT0[-31454] := B#16#0;
   STAT0[-31453] := B#16#0;
   STAT0[-31452] := B#16#0;
   STAT0[-31451] := B#16#0;
   STAT0[-31450] := B#16#0;
   STAT0[-31449] := B#16#0;
   STAT0[-31448] := B#16#0;
   STAT0[-31447] := B#16#0;
   STAT0[-31446] := B#16#0;
   STAT0[-31445] := B#16#1;
   STAT0[-31444] := B#16#0;
   STAT0[-31443] := B#16#0;
   STAT0[-31442] := B#16#0;
   STAT0[-31441] := B#16#0;
   STAT0[-31440] := B#16#0;
   STAT0[-31439] := B#16#0;
   STAT0[-31438] := B#16#0;
   STAT0[-31437] := B#16#0;
   STAT0[-31436] := B#16#0;
   STAT0[-31435] := B#16#0;
   STAT0[-31434] := B#16#0;
   STAT0[-31433] := B#16#0;
   STAT0[-31432] := B#16#0;
   STAT0[-31431] := B#16#0;
   STAT0[-31430] := B#16#0;
   STAT0[-31429] := B#16#0;
   STAT0[-31428] := B#16#0;
   STAT0[-31427] := B#16#0;
   STAT0[-31426] := B#16#0;
   STAT0[-31425] := B#16#0;
   STAT0[-31424] := B#16#0;
   STAT0[-31423] := B#16#0;
   STAT0[-31422] := B#16#0;
   STAT0[-31421] := B#16#0;
   STAT0[-31420] := B#16#0;
   STAT0[-31419] := B#16#0;
   STAT0[-31418] := B#16#0;
   STAT0[-31417] := B#16#0;
   STAT0[-31416] := B#16#0;
   STAT0[-31415] := B#16#0;
   STAT0[-31414] := B#16#0;
   STAT0[-31413] := B#16#0;
   STAT0[-31412] := B#16#0;
   STAT0[-31411] := B#16#0;
   STAT0[-31410] := B#16#0;
   STAT0[-31409] := B#16#0;
   STAT0[-31408] := B#16#0;
   STAT0[-31407] := B#16#0;
   STAT0[-31406] := B#16#0;
   STAT0[-31405] := B#16#0;
   STAT0[-31404] := B#16#0;
   STAT0[-31403] := B#16#0;
   STAT0[-31402] := B#16#0;
   STAT0[-31401] := B#16#0;
   STAT0[-31400] := B#16#0;
   STAT0[-31399] := B#16#0;
   STAT0[-31398] := B#16#0;
   STAT0[-31397] := B#16#0;
   STAT0[-31396] := B#16#0;
   STAT0[-31395] := B#16#0;
   STAT0[-31394] := B#16#0;
   STAT0[-31393] := B#16#0;
   STAT0[-31392] := B#16#0;
   STAT0[-31391] := B#16#0;
   STAT0[-31390] := B#16#0;
   STAT0[-31389] := B#16#0;
   STAT0[-31388] := B#16#0;
   STAT0[-31387] := B#16#0;
   STAT0[-31386] := B#16#0;
   STAT0[-31385] := B#16#0;
   STAT0[-31384] := B#16#0;
   STAT0[-31383] := B#16#0;
   STAT0[-31382] := B#16#0;
   STAT0[-31381] := B#16#0;
   STAT0[-31380] := B#16#0;
   STAT0[-31379] := B#16#0;
   STAT0[-31378] := B#16#0;
   STAT0[-31377] := B#16#0;
   STAT0[-31376] := B#16#0;
   STAT0[-31375] := B#16#0;
   STAT0[-31374] := B#16#0;
   STAT0[-31373] := B#16#0;
   STAT0[-31372] := B#16#0;
   STAT0[-31371] := B#16#0;
   STAT0[-31370] := B#16#0;
   STAT0[-31369] := B#16#0;
   STAT0[-31368] := B#16#0;
   STAT0[-31367] := B#16#0;
   STAT0[-31366] := B#16#0;
   STAT0[-31365] := B#16#0;
   STAT0[-31364] := B#16#0;
   STAT0[-31363] := B#16#0;
   STAT0[-31362] := B#16#0;
   STAT0[-31361] := B#16#0;
   STAT0[-31360] := B#16#0;
   STAT0[-31359] := B#16#0;
   STAT0[-31358] := B#16#0;
   STAT0[-31357] := B#16#0;
   STAT0[-31356] := B#16#0;
   STAT0[-31355] := B#16#0;
   STAT0[-31354] := B#16#0;
   STAT0[-31353] := B#16#0;
   STAT0[-31352] := B#16#0;
   STAT0[-31351] := B#16#0;
   STAT0[-31350] := B#16#0;
   STAT0[-31349] := B#16#0;
   STAT0[-31348] := B#16#0;
   STAT0[-31347] := B#16#0;
   STAT0[-31346] := B#16#0;
   STAT0[-31345] := B#16#0;
   STAT0[-31344] := B#16#0;
   STAT0[-31343] := B#16#0;
   STAT0[-31342] := B#16#0;
   STAT0[-31341] := B#16#0;
   STAT0[-31340] := B#16#0;
   STAT0[-31339] := B#16#0;
   STAT0[-31338] := B#16#0;
   STAT0[-31337] := B#16#0;
   STAT0[-31336] := B#16#0;
   STAT0[-31335] := B#16#0;
   STAT0[-31334] := B#16#0;
   STAT0[-31333] := B#16#0;
   STAT0[-31332] := B#16#0;
   STAT0[-31331] := B#16#0;
   STAT0[-31330] := B#16#0;
   STAT0[-31329] := B#16#0;
   STAT0[-31328] := B#16#0;
   STAT0[-31327] := B#16#0;
   STAT0[-31326] := B#16#0;
   STAT0[-31325] := B#16#0;
   STAT0[-31324] := B#16#0;
   STAT0[-31323] := B#16#0;
   STAT0[-31322] := B#16#0;
   STAT0[-31321] := B#16#0;
   STAT0[-31320] := B#16#0;
   STAT0[-31319] := B#16#0;
   STAT0[-31318] := B#16#0;
   STAT0[-31317] := B#16#0;
   STAT0[-31316] := B#16#0;
   STAT0[-31315] := B#16#0;
   STAT0[-31314] := B#16#0;
   STAT0[-31313] := B#16#0;
   STAT0[-31312] := B#16#0;
   STAT0[-31311] := B#16#0;
   STAT0[-31310] := B#16#0;
   STAT0[-31309] := B#16#0;
   STAT0[-31308] := B#16#0;
   STAT0[-31307] := B#16#0;
   STAT0[-31306] := B#16#0;
   STAT0[-31305] := B#16#0;
   STAT0[-31304] := B#16#0;
   STAT0[-31303] := B#16#0;
   STAT0[-31302] := B#16#0;
   STAT0[-31301] := B#16#0;
   STAT0[-31300] := B#16#0;
   STAT0[-31299] := B#16#0;
   STAT0[-31298] := B#16#0;
   STAT0[-31297] := B#16#0;
   STAT0[-31296] := B#16#0;
   STAT0[-31295] := B#16#0;
   STAT0[-31294] := B#16#0;
   STAT0[-31293] := B#16#0;
   STAT0[-31292] := B#16#0;
   STAT0[-31291] := B#16#0;
   STAT0[-31290] := B#16#0;
   STAT0[-31289] := B#16#0;
   STAT0[-31288] := B#16#0;
   STAT0[-31287] := B#16#0;
   STAT0[-31286] := B#16#0;
   STAT0[-31285] := B#16#0;
   STAT0[-31284] := B#16#0;
   STAT0[-31283] := B#16#0;
   STAT0[-31282] := B#16#0;
   STAT0[-31281] := B#16#0;
   STAT0[-31280] := B#16#0;
   STAT0[-31279] := B#16#0;
   STAT0[-31278] := B#16#0;
   STAT0[-31277] := B#16#0;
   STAT0[-31276] := B#16#0;
   STAT0[-31275] := B#16#0;
   STAT0[-31274] := B#16#0;
   STAT0[-31273] := B#16#0;
   STAT0[-31272] := B#16#0;
   STAT0[-31271] := B#16#0;
   STAT0[-31270] := B#16#0;
   STAT0[-31269] := B#16#0;
   STAT0[-31268] := B#16#0;
   STAT0[-31267] := B#16#0;
   STAT0[-31266] := B#16#0;
   STAT0[-31265] := B#16#0;
   STAT0[-31264] := B#16#0;
   STAT0[-31263] := B#16#0;
   STAT0[-31262] := B#16#0;
   STAT0[-31261] := B#16#0;
   STAT0[-31260] := B#16#0;
   STAT0[-31259] := B#16#0;
   STAT0[-31258] := B#16#0;
   STAT0[-31257] := B#16#0;
   STAT0[-31256] := B#16#0;
   STAT0[-31255] := B#16#0;
   STAT0[-31254] := B#16#0;
   STAT0[-31253] := B#16#0;
   STAT0[-31252] := B#16#0;
   STAT0[-31251] := B#16#0;
   STAT0[-31250] := B#16#0;
   STAT0[-31249] := B#16#0;
   STAT0[-31248] := B#16#0;
   STAT0[-31247] := B#16#0;
   STAT0[-31246] := B#16#0;
   STAT0[-31245] := B#16#0;
   STAT0[-31244] := B#16#0;
   STAT0[-31243] := B#16#0;
   STAT0[-31242] := B#16#0;
   STAT0[-31241] := B#16#0;
   STAT0[-31240] := B#16#0;
   STAT0[-31239] := B#16#0;
   STAT0[-31238] := B#16#0;
   STAT0[-31237] := B#16#0;
   STAT0[-31236] := B#16#0;
   STAT0[-31235] := B#16#0;
   STAT0[-31234] := B#16#0;
   STAT0[-31233] := B#16#0;
   STAT0[-31232] := B#16#0;
   STAT0[-31231] := B#16#0;
   STAT0[-31230] := B#16#0;
   STAT0[-31229] := B#16#0;
   STAT0[-31228] := B#16#0;
   STAT0[-31227] := B#16#0;
   STAT0[-31226] := B#16#0;
   STAT0[-31225] := B#16#0;
   STAT0[-31224] := B#16#0;
   STAT0[-31223] := B#16#0;
   STAT0[-31222] := B#16#0;
   STAT0[-31221] := B#16#0;
   STAT0[-31220] := B#16#0;
   STAT0[-31219] := B#16#0;
   STAT0[-31218] := B#16#0;
   STAT0[-31217] := B#16#0;
   STAT0[-31216] := B#16#0;
   STAT0[-31215] := B#16#0;
   STAT0[-31214] := B#16#0;
   STAT0[-31213] := B#16#0;
   STAT0[-31212] := B#16#0;
   STAT0[-31211] := B#16#0;
   STAT0[-31210] := B#16#0;
   STAT0[-31209] := B#16#0;
   STAT0[-31208] := B#16#0;
   STAT0[-31207] := B#16#0;
   STAT0[-31206] := B#16#0;
   STAT0[-31205] := B#16#0;
   STAT0[-31204] := B#16#0;
   STAT0[-31203] := B#16#0;
   STAT0[-31202] := B#16#0;
   STAT0[-31201] := B#16#0;
   STAT0[-31200] := B#16#0;
   STAT0[-31199] := B#16#0;
   STAT0[-31198] := B#16#0;
   STAT0[-31197] := B#16#0;
   STAT0[-31196] := B#16#0;
   STAT0[-31195] := B#16#0;
   STAT0[-31194] := B#16#0;
   STAT0[-31193] := B#16#0;
   STAT0[-31192] := B#16#0;
   STAT0[-31191] := B#16#0;
   STAT0[-31190] := B#16#0;
   STAT0[-31189] := B#16#0;
   STAT0[-31188] := B#16#0;
   STAT0[-31187] := B#16#0;
   STAT0[-31186] := B#16#0;
   STAT0[-31185] := B#16#0;
   STAT0[-31184] := B#16#0;
   STAT0[-31183] := B#16#0;
   STAT0[-31182] := B#16#0;
   STAT0[-31181] := B#16#0;
   STAT0[-31180] := B#16#0;
   STAT0[-31179] := B#16#0;
   STAT0[-31178] := B#16#0;
   STAT0[-31177] := B#16#0;
   STAT0[-31176] := B#16#0;
   STAT0[-31175] := B#16#0;
   STAT0[-31174] := B#16#0;
   STAT0[-31173] := B#16#0;
   STAT0[-31172] := B#16#0;
   STAT0[-31171] := B#16#0;
   STAT0[-31170] := B#16#0;
   STAT0[-31169] := B#16#0;
   STAT0[-31168] := B#16#0;
   STAT0[-31167] := B#16#0;
   STAT0[-31166] := B#16#0;
   STAT0[-31165] := B#16#0;
   STAT0[-31164] := B#16#0;
   STAT0[-31163] := B#16#0;
   STAT0[-31162] := B#16#0;
   STAT0[-31161] := B#16#0;
   STAT0[-31160] := B#16#0;
   STAT0[-31159] := B#16#0;
   STAT0[-31158] := B#16#0;
   STAT0[-31157] := B#16#0;
   STAT0[-31156] := B#16#0;
   STAT0[-31155] := B#16#0;
   STAT0[-31154] := B#16#0;
   STAT0[-31153] := B#16#0;
   STAT0[-31152] := B#16#0;
   STAT0[-31151] := B#16#0;
   STAT0[-31150] := B#16#0;
   STAT0[-31149] := B#16#0;
   STAT0[-31148] := B#16#0;
   STAT0[-31147] := B#16#0;
   STAT0[-31146] := B#16#0;
   STAT0[-31145] := B#16#0;
   STAT0[-31144] := B#16#0;
   STAT0[-31143] := B#16#0;
   STAT0[-31142] := B#16#0;
   STAT0[-31141] := B#16#0;
   STAT0[-31140] := B#16#0;
   STAT0[-31139] := B#16#0;
   STAT0[-31138] := B#16#0;
   STAT0[-31137] := B#16#0;
   STAT0[-31136] := B#16#0;
   STAT0[-31135] := B#16#0;
   STAT0[-31134] := B#16#0;
   STAT0[-31133] := B#16#0;
   STAT0[-31132] := B#16#0;
   STAT0[-31131] := B#16#0;
   STAT0[-31130] := B#16#0;
   STAT0[-31129] := B#16#0;
   STAT0[-31128] := B#16#0;
   STAT0[-31127] := B#16#0;
   STAT0[-31126] := B#16#0;
   STAT0[-31125] := B#16#0;
   STAT0[-31124] := B#16#0;
   STAT0[-31123] := B#16#0;
   STAT0[-31122] := B#16#0;
   STAT0[-31121] := B#16#0;
   STAT0[-31120] := B#16#0;
   STAT0[-31119] := B#16#0;
   STAT0[-31118] := B#16#0;
   STAT0[-31117] := B#16#0;
   STAT0[-31116] := B#16#0;
   STAT0[-31115] := B#16#0;
   STAT0[-31114] := B#16#0;
   STAT0[-31113] := B#16#0;
   STAT0[-31112] := B#16#0;
   STAT0[-31111] := B#16#0;
   STAT0[-31110] := B#16#0;
   STAT0[-31109] := B#16#0;
   STAT0[-31108] := B#16#0;
   STAT0[-31107] := B#16#0;
   STAT0[-31106] := B#16#0;
   STAT0[-31105] := B#16#0;
   STAT0[-31104] := B#16#0;
   STAT0[-31103] := B#16#0;
   STAT0[-31102] := B#16#0;
   STAT0[-31101] := B#16#0;
   STAT0[-31100] := B#16#0;
   STAT0[-31099] := B#16#0;
   STAT0[-31098] := B#16#0;
   STAT0[-31097] := B#16#0;
   STAT0[-31096] := B#16#0;
   STAT0[-31095] := B#16#0;
   STAT0[-31094] := B#16#0;
   STAT0[-31093] := B#16#0;
   STAT0[-31092] := B#16#0;
   STAT0[-31091] := B#16#0;
   STAT0[-31090] := B#16#0;
   STAT0[-31089] := B#16#0;
   STAT0[-31088] := B#16#0;
   STAT0[-31087] := B#16#0;
   STAT0[-31086] := B#16#0;
   STAT0[-31085] := B#16#0;
   STAT0[-31084] := B#16#0;
   STAT0[-31083] := B#16#0;
   STAT0[-31082] := B#16#0;
   STAT0[-31081] := B#16#0;
   STAT0[-31080] := B#16#0;
   STAT0[-31079] := B#16#0;
   STAT0[-31078] := B#16#0;
   STAT0[-31077] := B#16#0;
   STAT0[-31076] := B#16#0;
   STAT0[-31075] := B#16#0;
   STAT0[-31074] := B#16#0;
   STAT0[-31073] := B#16#0;
   STAT0[-31072] := B#16#0;
   STAT0[-31071] := B#16#0;
   STAT0[-31070] := B#16#0;
   STAT0[-31069] := B#16#0;
   STAT0[-31068] := B#16#0;
   STAT0[-31067] := B#16#0;
   STAT0[-31066] := B#16#0;
   STAT0[-31065] := B#16#0;
   STAT0[-31064] := B#16#0;
   STAT0[-31063] := B#16#0;
   STAT0[-31062] := B#16#0;
   STAT0[-31061] := B#16#0;
   STAT0[-31060] := B#16#0;
   STAT0[-31059] := B#16#0;
   STAT0[-31058] := B#16#0;
   STAT0[-31057] := B#16#0;
   STAT0[-31056] := B#16#0;
   STAT0[-31055] := B#16#0;
   STAT0[-31054] := B#16#0;
   STAT0[-31053] := B#16#0;
   STAT0[-31052] := B#16#0;
   STAT0[-31051] := B#16#0;
   STAT0[-31050] := B#16#0;
   STAT0[-31049] := B#16#0;
   STAT0[-31048] := B#16#0;
   STAT0[-31047] := B#16#0;
   STAT0[-31046] := B#16#0;
   STAT0[-31045] := B#16#0;
   STAT0[-31044] := B#16#0;
   STAT0[-31043] := B#16#0;
   STAT0[-31042] := B#16#0;
   STAT0[-31041] := B#16#0;
   STAT0[-31040] := B#16#0;
   STAT0[-31039] := B#16#0;
   STAT0[-31038] := B#16#0;
   STAT0[-31037] := B#16#0;
   STAT0[-31036] := B#16#0;
   STAT0[-31035] := B#16#0;
   STAT0[-31034] := B#16#0;
   STAT0[-31033] := B#16#0;
   STAT0[-31032] := B#16#0;
   STAT0[-31031] := B#16#0;
   STAT0[-31030] := B#16#0;
   STAT0[-31029] := B#16#0;
   STAT0[-31028] := B#16#0;
   STAT0[-31027] := B#16#0;
   STAT0[-31026] := B#16#0;
   STAT0[-31025] := B#16#0;
   STAT0[-31024] := B#16#0;
   STAT0[-31023] := B#16#0;
   STAT0[-31022] := B#16#0;
   STAT0[-31021] := B#16#0;
   STAT0[-31020] := B#16#0;
   STAT0[-31019] := B#16#0;
   STAT0[-31018] := B#16#0;
   STAT0[-31017] := B#16#0;
   STAT0[-31016] := B#16#0;
   STAT0[-31015] := B#16#0;
   STAT0[-31014] := B#16#0;
   STAT0[-31013] := B#16#0;
   STAT0[-31012] := B#16#0;
   STAT0[-31011] := B#16#0;
   STAT0[-31010] := B#16#0;
   STAT0[-31009] := B#16#0;
   STAT0[-31008] := B#16#0;
   STAT0[-31007] := B#16#0;
   STAT0[-31006] := B#16#0;
   STAT0[-31005] := B#16#0;
   STAT0[-31004] := B#16#0;
   STAT0[-31003] := B#16#0;
   STAT0[-31002] := B#16#0;
   STAT0[-31001] := B#16#0;
   STAT0[-31000] := B#16#0;
   STAT0[-30999] := B#16#0;
   STAT0[-30998] := B#16#0;
   STAT0[-30997] := B#16#0;
   STAT0[-30996] := B#16#0;
   STAT0[-30995] := B#16#0;
   STAT0[-30994] := B#16#0;
   STAT0[-30993] := B#16#0;
   STAT0[-30992] := B#16#0;
   STAT0[-30991] := B#16#0;
   STAT0[-30990] := B#16#0;
   STAT0[-30989] := B#16#0;
   STAT0[-30988] := B#16#0;
   STAT0[-30987] := B#16#0;
   STAT0[-30986] := B#16#0;
   STAT0[-30985] := B#16#0;
   STAT0[-30984] := B#16#0;
   STAT0[-30983] := B#16#0;
   STAT0[-30982] := B#16#0;
   STAT0[-30981] := B#16#0;
   STAT0[-30980] := B#16#0;
   STAT0[-30979] := B#16#0;
   STAT0[-30978] := B#16#0;
   STAT0[-30977] := B#16#0;
   STAT0[-30976] := B#16#0;
   STAT0[-30975] := B#16#0;
   STAT0[-30974] := B#16#0;
   STAT0[-30973] := B#16#0;
   STAT0[-30972] := B#16#0;
   STAT0[-30971] := B#16#0;
   STAT0[-30970] := B#16#0;
   STAT0[-30969] := B#16#0;
   STAT0[-30968] := B#16#0;
   STAT0[-30967] := B#16#0;
   STAT0[-30966] := B#16#0;
   STAT0[-30965] := B#16#0;
   STAT0[-30964] := B#16#0;
   STAT0[-30963] := B#16#0;
   STAT0[-30962] := B#16#0;
   STAT0[-30961] := B#16#0;
   STAT0[-30960] := B#16#0;
   STAT0[-30959] := B#16#0;
   STAT0[-30958] := B#16#0;
   STAT0[-30957] := B#16#0;
   STAT0[-30956] := B#16#0;
   STAT0[-30955] := B#16#0;
   STAT0[-30954] := B#16#0;
   STAT0[-30953] := B#16#0;
   STAT0[-30952] := B#16#0;
   STAT0[-30951] := B#16#0;
   STAT0[-30950] := B#16#0;
   STAT0[-30949] := B#16#0;
   STAT0[-30948] := B#16#0;
   STAT0[-30947] := B#16#0;
   STAT0[-30946] := B#16#0;
   STAT0[-30945] := B#16#0;
   STAT0[-30944] := B#16#0;
   STAT0[-30943] := B#16#0;
   STAT0[-30942] := B#16#0;
   STAT0[-30941] := B#16#0;
   STAT0[-30940] := B#16#0;
   STAT0[-30939] := B#16#0;
   STAT0[-30938] := B#16#0;
   STAT0[-30937] := B#16#0;
   STAT0[-30936] := B#16#0;
   STAT0[-30935] := B#16#0;
   STAT0[-30934] := B#16#0;
   STAT0[-30933] := B#16#0;
   STAT0[-30932] := B#16#0;
   STAT0[-30931] := B#16#0;
   STAT0[-30930] := B#16#0;
   STAT0[-30929] := B#16#0;
   STAT0[-30928] := B#16#0;
   STAT0[-30927] := B#16#0;
   STAT0[-30926] := B#16#0;
   STAT0[-30925] := B#16#0;
   STAT0[-30924] := B#16#0;
   STAT0[-30923] := B#16#0;
   STAT0[-30922] := B#16#0;
   STAT0[-30921] := B#16#0;
   STAT0[-30920] := B#16#0;
   STAT0[-30919] := B#16#0;
   STAT0[-30918] := B#16#0;
   STAT0[-30917] := B#16#0;
   STAT0[-30916] := B#16#0;
   STAT0[-30915] := B#16#0;
   STAT0[-30914] := B#16#0;
   STAT0[-30913] := B#16#0;
   STAT0[-30912] := B#16#0;
   STAT0[-30911] := B#16#0;
   STAT0[-30910] := B#16#0;
   STAT0[-30909] := B#16#0;
   STAT0[-30908] := B#16#0;
   STAT0[-30907] := B#16#0;
   STAT0[-30906] := B#16#0;
   STAT0[-30905] := B#16#0;
   STAT0[-30904] := B#16#0;
   STAT0[-30903] := B#16#0;
   STAT0[-30902] := B#16#0;
   STAT0[-30901] := B#16#0;
   STAT0[-30900] := B#16#0;
   STAT0[-30899] := B#16#0;
   STAT0[-30898] := B#16#0;
   STAT0[-30897] := B#16#0;
   STAT0[-30896] := B#16#0;
   STAT0[-30895] := B#16#0;
   STAT0[-30894] := B#16#0;
   STAT0[-30893] := B#16#0;
   STAT0[-30892] := B#16#0;
   STAT0[-30891] := B#16#0;
   STAT0[-30890] := B#16#0;
   STAT0[-30889] := B#16#0;
   STAT0[-30888] := B#16#0;
   STAT0[-30887] := B#16#0;
   STAT0[-30886] := B#16#0;
   STAT0[-30885] := B#16#0;
   STAT0[-30884] := B#16#0;
   STAT0[-30883] := B#16#0;
   STAT0[-30882] := B#16#0;
   STAT0[-30881] := B#16#0;
   STAT0[-30880] := B#16#0;
   STAT0[-30879] := B#16#0;
   STAT0[-30878] := B#16#0;
   STAT0[-30877] := B#16#0;
   STAT0[-30876] := B#16#0;
   STAT0[-30875] := B#16#0;
   STAT0[-30874] := B#16#0;
   STAT0[-30873] := B#16#0;
   STAT0[-30872] := B#16#0;
   STAT0[-30871] := B#16#0;
   STAT0[-30870] := B#16#0;
   STAT0[-30869] := B#16#0;
   STAT0[-30868] := B#16#0;
   STAT0[-30867] := B#16#0;
   STAT0[-30866] := B#16#0;
   STAT0[-30865] := B#16#0;
   STAT0[-30864] := B#16#0;
   STAT0[-30863] := B#16#0;
   STAT0[-30862] := B#16#0;
   STAT0[-30861] := B#16#0;
   STAT0[-30860] := B#16#0;
   STAT0[-30859] := B#16#0;
   STAT0[-30858] := B#16#0;
   STAT0[-30857] := B#16#0;
   STAT0[-30856] := B#16#0;
   STAT0[-30855] := B#16#0;
   STAT0[-30854] := B#16#0;
   STAT0[-30853] := B#16#0;
   STAT0[-30852] := B#16#0;
   STAT0[-30851] := B#16#0;
   STAT0[-30850] := B#16#0;
   STAT0[-30849] := B#16#0;
   STAT0[-30848] := B#16#0;
   STAT0[-30847] := B#16#0;
   STAT0[-30846] := B#16#0;
   STAT0[-30845] := B#16#0;
   STAT0[-30844] := B#16#0;
   STAT0[-30843] := B#16#0;
   STAT0[-30842] := B#16#0;
   STAT0[-30841] := B#16#0;
   STAT0[-30840] := B#16#0;
   STAT0[-30839] := B#16#0;
   STAT0[-30838] := B#16#0;
   STAT0[-30837] := B#16#0;
   STAT0[-30836] := B#16#0;
   STAT0[-30835] := B#16#0;
   STAT0[-30834] := B#16#0;
   STAT0[-30833] := B#16#0;
   STAT0[-30832] := B#16#0;
   STAT0[-30831] := B#16#0;
   STAT0[-30830] := B#16#0;
   STAT0[-30829] := B#16#0;
   STAT0[-30828] := B#16#0;
   STAT0[-30827] := B#16#0;
   STAT0[-30826] := B#16#0;
   STAT0[-30825] := B#16#0;
   STAT0[-30824] := B#16#0;
   STAT0[-30823] := B#16#0;
   STAT0[-30822] := B#16#0;
   STAT0[-30821] := B#16#0;
   STAT0[-30820] := B#16#0;
   STAT0[-30819] := B#16#0;
   STAT0[-30818] := B#16#0;
   STAT0[-30817] := B#16#0;
   STAT0[-30816] := B#16#0;
   STAT0[-30815] := B#16#0;
   STAT0[-30814] := B#16#0;
   STAT0[-30813] := B#16#0;
   STAT0[-30812] := B#16#0;
   STAT0[-30811] := B#16#0;
   STAT0[-30810] := B#16#0;
   STAT0[-30809] := B#16#0;
   STAT0[-30808] := B#16#0;
   STAT0[-30807] := B#16#0;
   STAT0[-30806] := B#16#0;
   STAT0[-30805] := B#16#0;
   STAT0[-30804] := B#16#0;
   STAT0[-30803] := B#16#0;
   STAT0[-30802] := B#16#0;
   STAT0[-30801] := B#16#0;
   STAT0[-30800] := B#16#0;
   STAT0[-30799] := B#16#0;
   STAT0[-30798] := B#16#0;
   STAT0[-30797] := B#16#0;
   STAT0[-30796] := B#16#0;
   STAT0[-30795] := B#16#0;
   STAT0[-30794] := B#16#0;
   STAT0[-30793] := B#16#0;
   STAT0[-30792] := B#16#0;
   STAT0[-30791] := B#16#0;
   STAT0[-30790] := B#16#0;
   STAT0[-30789] := B#16#0;
   STAT0[-30788] := B#16#0;
   STAT0[-30787] := B#16#0;
   STAT0[-30786] := B#16#0;
   STAT0[-30785] := B#16#0;
   STAT0[-30784] := B#16#0;
   STAT0[-30783] := B#16#0;
   STAT0[-30782] := B#16#0;
   STAT0[-30781] := B#16#0;
   STAT0[-30780] := B#16#0;
   STAT0[-30779] := B#16#0;
   STAT0[-30778] := B#16#0;
   STAT0[-30777] := B#16#0;
   STAT0[-30776] := B#16#0;
   STAT0[-30775] := B#16#0;
   STAT0[-30774] := B#16#0;
   STAT0[-30773] := B#16#0;
   STAT0[-30772] := B#16#0;
   STAT0[-30771] := B#16#0;
   STAT0[-30770] := B#16#0;
   STAT0[-30769] := B#16#0;
   STAT0[-30768] := B#16#0;
   STAT0[-30767] := B#16#0;
   STAT0[-30766] := B#16#0;
   STAT0[-30765] := B#16#0;
   STAT0[-30764] := B#16#0;
   STAT0[-30763] := B#16#0;
   STAT0[-30762] := B#16#0;
   STAT0[-30761] := B#16#0;
   STAT0[-30760] := B#16#0;
   STAT0[-30759] := B#16#0;
   STAT0[-30758] := B#16#0;
   STAT0[-30757] := B#16#0;
   STAT0[-30756] := B#16#0;
   STAT0[-30755] := B#16#0;
   STAT0[-30754] := B#16#0;
   STAT0[-30753] := B#16#0;
   STAT0[-30752] := B#16#0;
   STAT0[-30751] := B#16#0;
   STAT0[-30750] := B#16#0;
   STAT0[-30749] := B#16#0;
   STAT0[-30748] := B#16#0;
   STAT0[-30747] := B#16#0;
   STAT0[-30746] := B#16#0;
   STAT0[-30745] := B#16#0;
   STAT0[-30744] := B#16#0;
   STAT0[-30743] := B#16#0;
   STAT0[-30742] := B#16#0;
   STAT0[-30741] := B#16#0;
   STAT0[-30740] := B#16#0;
   STAT0[-30739] := B#16#0;
   STAT0[-30738] := B#16#0;
   STAT0[-30737] := B#16#0;
   STAT0[-30736] := B#16#0;
   STAT0[-30735] := B#16#0;
   STAT0[-30734] := B#16#0;
   STAT0[-30733] := B#16#0;
   STAT0[-30732] := B#16#0;
   STAT0[-30731] := B#16#0;
   STAT0[-30730] := B#16#0;
   STAT0[-30729] := B#16#0;
   STAT0[-30728] := B#16#0;
   STAT0[-30727] := B#16#0;
   STAT0[-30726] := B#16#0;
   STAT0[-30725] := B#16#0;
   STAT0[-30724] := B#16#0;
   STAT0[-30723] := B#16#0;
   STAT0[-30722] := B#16#0;
   STAT0[-30721] := B#16#0;
   STAT0[-30720] := B#16#90;
   STAT0[-30719] := B#16#1;
   STAT0[-30718] := B#16#1;
   STAT0[-30717] := B#16#0;
   STAT0[-30716] := B#16#0;
   STAT0[-30715] := B#16#0;
   STAT0[-30714] := B#16#0;
   STAT0[-30713] := B#16#2;
   STAT0[-30712] := B#16#0;
   STAT0[-30711] := B#16#0;
   STAT0[-30710] := B#16#0;
   STAT0[-30709] := B#16#0;
   STAT0[-30708] := B#16#0;
   STAT0[-30707] := B#16#0;
   STAT0[-30706] := B#16#0;
   STAT0[-30705] := B#16#0;
   STAT0[-30704] := B#16#0;
   STAT0[-30703] := B#16#0;
   STAT0[-30702] := B#16#0;
   STAT0[-30701] := B#16#0;
   STAT0[-30700] := B#16#0;
   STAT0[-30699] := B#16#0;
   STAT0[-30698] := B#16#0;
   STAT0[-30697] := B#16#0;
   STAT0[-30696] := B#16#0;
   STAT0[-30695] := B#16#0;
   STAT0[-30694] := B#16#0;
   STAT0[-30693] := B#16#0;
   STAT0[-30692] := B#16#0;
   STAT0[-30691] := B#16#0;
   STAT0[-30690] := B#16#0;
   STAT0[-30689] := B#16#0;
   STAT0[-30688] := B#16#0;
   STAT0[-30687] := B#16#0;
   STAT0[-30686] := B#16#0;
   STAT0[-30685] := B#16#0;
   STAT0[-30684] := B#16#0;
   STAT0[-30683] := B#16#0;
   STAT0[-30682] := B#16#0;
   STAT0[-30681] := B#16#0;
   STAT0[-30680] := B#16#0;
   STAT0[-30679] := B#16#0;
   STAT0[-30678] := B#16#0;
   STAT0[-30677] := B#16#0;
   STAT0[-30676] := B#16#0;
   STAT0[-30675] := B#16#0;
   STAT0[-30674] := B#16#0;
   STAT0[-30673] := B#16#0;
   STAT0[-30672] := B#16#0;
   STAT0[-30671] := B#16#0;
   STAT0[-30670] := B#16#0;
   STAT0[-30669] := B#16#0;
   STAT0[-30668] := B#16#0;
   STAT0[-30667] := B#16#0;
   STAT0[-30666] := B#16#0;
   STAT0[-30665] := B#16#0;
   STAT0[-30664] := B#16#0;
   STAT0[-30663] := B#16#0;
   STAT0[-30662] := B#16#0;
   STAT0[-30661] := B#16#0;
   STAT0[-30660] := B#16#0;
   STAT0[-30659] := B#16#0;
   STAT0[-30658] := B#16#0;
   STAT0[-30657] := B#16#0;
   STAT0[-30656] := B#16#0;
   STAT0[-30655] := B#16#0;
   STAT0[-30654] := B#16#0;
   STAT0[-30653] := B#16#0;
   STAT0[-30652] := B#16#0;
   STAT0[-30651] := B#16#0;
   STAT0[-30650] := B#16#0;
   STAT0[-30649] := B#16#0;
   STAT0[-30648] := B#16#0;
   STAT0[-30647] := B#16#0;
   STAT0[-30646] := B#16#0;
   STAT0[-30645] := B#16#0;
   STAT0[-30644] := B#16#0;
   STAT0[-30643] := B#16#0;
   STAT0[-30642] := B#16#0;
   STAT0[-30641] := B#16#0;
   STAT0[-30640] := B#16#0;
   STAT0[-30639] := B#16#0;
   STAT0[-30638] := B#16#0;
   STAT0[-30637] := B#16#0;
   STAT0[-30636] := B#16#0;
   STAT0[-30635] := B#16#0;
   STAT0[-30634] := B#16#0;
   STAT0[-30633] := B#16#0;
   STAT0[-30632] := B#16#0;
   STAT0[-30631] := B#16#0;
   STAT0[-30630] := B#16#0;
   STAT0[-30629] := B#16#0;
   STAT0[-30628] := B#16#0;
   STAT0[-30627] := B#16#0;
   STAT0[-30626] := B#16#0;
   STAT0[-30625] := B#16#0;
   STAT0[-30624] := B#16#0;
   STAT0[-30623] := B#16#0;
   STAT0[-30622] := B#16#0;
   STAT0[-30621] := B#16#0;
   STAT0[-30620] := B#16#0;
   STAT0[-30619] := B#16#0;
   STAT0[-30618] := B#16#0;
   STAT0[-30617] := B#16#0;
   STAT0[-30616] := B#16#0;
   STAT0[-30615] := B#16#0;
   STAT0[-30614] := B#16#0;
   STAT0[-30613] := B#16#0;
   STAT0[-30612] := B#16#0;
   STAT0[-30611] := B#16#0;
   STAT0[-30610] := B#16#0;
   STAT0[-30609] := B#16#0;
   STAT0[-30608] := B#16#0;
   STAT0[-30607] := B#16#0;
   STAT0[-30606] := B#16#0;
   STAT0[-30605] := B#16#0;
   STAT0[-30604] := B#16#0;
   STAT0[-30603] := B#16#0;
   STAT0[-30602] := B#16#0;
   STAT0[-30601] := B#16#0;
   STAT0[-30600] := B#16#0;
   STAT0[-30599] := B#16#0;
   STAT0[-30598] := B#16#0;
   STAT0[-30597] := B#16#0;
   STAT0[-30596] := B#16#0;
   STAT0[-30595] := B#16#0;
   STAT0[-30594] := B#16#0;
   STAT0[-30593] := B#16#0;
   STAT0[-30592] := B#16#0;
   STAT0[-30591] := B#16#0;
   STAT0[-30590] := B#16#0;
   STAT0[-30589] := B#16#0;
   STAT0[-30588] := B#16#0;
   STAT0[-30587] := B#16#0;
   STAT0[-30586] := B#16#0;
   STAT0[-30585] := B#16#0;
   STAT0[-30584] := B#16#0;
   STAT0[-30583] := B#16#0;
   STAT0[-30582] := B#16#0;
   STAT0[-30581] := B#16#0;
   STAT0[-30580] := B#16#0;
   STAT0[-30579] := B#16#0;
   STAT0[-30578] := B#16#0;
   STAT0[-30577] := B#16#0;
   STAT0[-30576] := B#16#0;
   STAT0[-30575] := B#16#0;
   STAT0[-30574] := B#16#0;
   STAT0[-30573] := B#16#0;
   STAT0[-30572] := B#16#0;
   STAT0[-30571] := B#16#0;
   STAT0[-30570] := B#16#0;
   STAT0[-30569] := B#16#0;
   STAT0[-30568] := B#16#0;
   STAT0[-30567] := B#16#0;
   STAT0[-30566] := B#16#0;
   STAT0[-30565] := B#16#0;
   STAT0[-30564] := B#16#0;
   STAT0[-30563] := B#16#0;
   STAT0[-30562] := B#16#0;
   STAT0[-30561] := B#16#0;
   STAT0[-30560] := B#16#0;
   STAT0[-30559] := B#16#0;
   STAT0[-30558] := B#16#0;
   STAT0[-30557] := B#16#0;
   STAT0[-30556] := B#16#0;
   STAT0[-30555] := B#16#0;
   STAT0[-30554] := B#16#0;
   STAT0[-30553] := B#16#0;
   STAT0[-30552] := B#16#0;
   STAT0[-30551] := B#16#0;
   STAT0[-30550] := B#16#0;
   STAT0[-30549] := B#16#0;
   STAT0[-30548] := B#16#0;
   STAT0[-30547] := B#16#0;
   STAT0[-30546] := B#16#0;
   STAT0[-30545] := B#16#0;
   STAT0[-30544] := B#16#0;
   STAT0[-30543] := B#16#0;
   STAT0[-30542] := B#16#0;
   STAT0[-30541] := B#16#0;
   STAT0[-30540] := B#16#0;
   STAT0[-30539] := B#16#0;
   STAT0[-30538] := B#16#0;
   STAT0[-30537] := B#16#0;
   STAT0[-30536] := B#16#0;
   STAT0[-30535] := B#16#0;
   STAT0[-30534] := B#16#0;
   STAT0[-30533] := B#16#0;
   STAT0[-30532] := B#16#0;
   STAT0[-30531] := B#16#0;
   STAT0[-30530] := B#16#0;
   STAT0[-30529] := B#16#0;
   STAT0[-30528] := B#16#0;
   STAT0[-30527] := B#16#0;
   STAT0[-30526] := B#16#0;
   STAT0[-30525] := B#16#0;
   STAT0[-30524] := B#16#0;
   STAT0[-30523] := B#16#0;
   STAT0[-30522] := B#16#0;
   STAT0[-30521] := B#16#0;
   STAT0[-30520] := B#16#0;
   STAT0[-30519] := B#16#0;
   STAT0[-30518] := B#16#0;
   STAT0[-30517] := B#16#0;
   STAT0[-30516] := B#16#0;
   STAT0[-30515] := B#16#0;
   STAT0[-30514] := B#16#0;
   STAT0[-30513] := B#16#0;
   STAT0[-30512] := B#16#0;
   STAT0[-30511] := B#16#0;
   STAT0[-30510] := B#16#0;
   STAT0[-30509] := B#16#0;
   STAT0[-30508] := B#16#0;
   STAT0[-30507] := B#16#0;
   STAT0[-30506] := B#16#0;
   STAT0[-30505] := B#16#0;
   STAT0[-30504] := B#16#0;
   STAT0[-30503] := B#16#0;
   STAT0[-30502] := B#16#0;
   STAT0[-30501] := B#16#0;
   STAT0[-30500] := B#16#0;
   STAT0[-30499] := B#16#0;
   STAT0[-30498] := B#16#0;
   STAT0[-30497] := B#16#0;
   STAT0[-30496] := B#16#0;
   STAT0[-30495] := B#16#0;
   STAT0[-30494] := B#16#0;
   STAT0[-30493] := B#16#0;
   STAT0[-30492] := B#16#0;
   STAT0[-30491] := B#16#0;
   STAT0[-30490] := B#16#0;
   STAT0[-30489] := B#16#0;
   STAT0[-30488] := B#16#0;
   STAT0[-30487] := B#16#0;
   STAT0[-30486] := B#16#0;
   STAT0[-30485] := B#16#0;
   STAT0[-30484] := B#16#0;
   STAT0[-30483] := B#16#0;
   STAT0[-30482] := B#16#0;
   STAT0[-30481] := B#16#0;
   STAT0[-30480] := B#16#0;
   STAT0[-30479] := B#16#0;
   STAT0[-30478] := B#16#0;
   STAT0[-30477] := B#16#0;
   STAT0[-30476] := B#16#0;
   STAT0[-30475] := B#16#0;
   STAT0[-30474] := B#16#0;
   STAT0[-30473] := B#16#0;
   STAT0[-30472] := B#16#0;
   STAT0[-30471] := B#16#0;
   STAT0[-30470] := B#16#0;
   STAT0[-30469] := B#16#0;
   STAT0[-30468] := B#16#0;
   STAT0[-30467] := B#16#0;
   STAT0[-30466] := B#16#0;
   STAT0[-30465] := B#16#0;
   STAT0[-30464] := B#16#0;
   STAT0[-30463] := B#16#0;
   STAT0[-30462] := B#16#0;
   STAT0[-30461] := B#16#0;
   STAT0[-30460] := B#16#0;
   STAT0[-30459] := B#16#0;
   STAT0[-30458] := B#16#0;
   STAT0[-30457] := B#16#0;
   STAT0[-30456] := B#16#0;
   STAT0[-30455] := B#16#0;
   STAT0[-30454] := B#16#0;
   STAT0[-30453] := B#16#0;
   STAT0[-30452] := B#16#0;
   STAT0[-30451] := B#16#0;
   STAT0[-30450] := B#16#0;
   STAT0[-30449] := B#16#0;
   STAT0[-30448] := B#16#0;
   STAT0[-30447] := B#16#0;
   STAT0[-30446] := B#16#0;
   STAT0[-30445] := B#16#0;
   STAT0[-30444] := B#16#0;
   STAT0[-30443] := B#16#0;
   STAT0[-30442] := B#16#0;
   STAT0[-30441] := B#16#0;
   STAT0[-30440] := B#16#0;
   STAT0[-30439] := B#16#0;
   STAT0[-30438] := B#16#0;
   STAT0[-30437] := B#16#0;
   STAT0[-30436] := B#16#0;
   STAT0[-30435] := B#16#0;
   STAT0[-30434] := B#16#0;
   STAT0[-30433] := B#16#0;
   STAT0[-30432] := B#16#0;
   STAT0[-30431] := B#16#0;
   STAT0[-30430] := B#16#0;
   STAT0[-30429] := B#16#0;
   STAT0[-30428] := B#16#0;
   STAT0[-30427] := B#16#0;
   STAT0[-30426] := B#16#0;
   STAT0[-30425] := B#16#0;
   STAT0[-30424] := B#16#0;
   STAT0[-30423] := B#16#0;
   STAT0[-30422] := B#16#0;
   STAT0[-30421] := B#16#0;
   STAT0[-30420] := B#16#0;
   STAT0[-30419] := B#16#0;
   STAT0[-30418] := B#16#0;
   STAT0[-30417] := B#16#0;
   STAT0[-30416] := B#16#0;
   STAT0[-30415] := B#16#0;
   STAT0[-30414] := B#16#0;
   STAT0[-30413] := B#16#0;
   STAT0[-30412] := B#16#0;
   STAT0[-30411] := B#16#0;
   STAT0[-30410] := B#16#0;
   STAT0[-30409] := B#16#0;
   STAT0[-30408] := B#16#0;
   STAT0[-30407] := B#16#0;
   STAT0[-30406] := B#16#0;
   STAT0[-30405] := B#16#0;
   STAT0[-30404] := B#16#0;
   STAT0[-30403] := B#16#0;
   STAT0[-30402] := B#16#0;
   STAT0[-30401] := B#16#0;
   STAT0[-30400] := B#16#0;
   STAT0[-30399] := B#16#0;
   STAT0[-30398] := B#16#0;
   STAT0[-30397] := B#16#0;
   STAT0[-30396] := B#16#0;
   STAT0[-30395] := B#16#0;
   STAT0[-30394] := B#16#0;
   STAT0[-30393] := B#16#0;
   STAT0[-30392] := B#16#0;
   STAT0[-30391] := B#16#0;
   STAT0[-30390] := B#16#0;
   STAT0[-30389] := B#16#0;
   STAT0[-30388] := B#16#0;
   STAT0[-30387] := B#16#0;
   STAT0[-30386] := B#16#0;
   STAT0[-30385] := B#16#0;
   STAT0[-30384] := B#16#0;
   STAT0[-30383] := B#16#0;
   STAT0[-30382] := B#16#0;
   STAT0[-30381] := B#16#0;
   STAT0[-30380] := B#16#0;
   STAT0[-30379] := B#16#0;
   STAT0[-30378] := B#16#0;
   STAT0[-30377] := B#16#0;
   STAT0[-30376] := B#16#0;
   STAT0[-30375] := B#16#0;
   STAT0[-30374] := B#16#0;
   STAT0[-30373] := B#16#0;
   STAT0[-30372] := B#16#0;
   STAT0[-30371] := B#16#0;
   STAT0[-30370] := B#16#0;
   STAT0[-30369] := B#16#0;
   STAT0[-30368] := B#16#0;
   STAT0[-30367] := B#16#0;
   STAT0[-30366] := B#16#0;
   STAT0[-30365] := B#16#0;
   STAT0[-30364] := B#16#0;
   STAT0[-30363] := B#16#0;
   STAT0[-30362] := B#16#0;
   STAT0[-30361] := B#16#0;
   STAT0[-30360] := B#16#0;
   STAT0[-30359] := B#16#0;
   STAT0[-30358] := B#16#0;
   STAT0[-30357] := B#16#0;
   STAT0[-30356] := B#16#0;
   STAT0[-30355] := B#16#0;
   STAT0[-30354] := B#16#0;
   STAT0[-30353] := B#16#0;
   STAT0[-30352] := B#16#0;
   STAT0[-30351] := B#16#0;
   STAT0[-30350] := B#16#0;
   STAT0[-30349] := B#16#0;
   STAT0[-30348] := B#16#0;
   STAT0[-30347] := B#16#0;
   STAT0[-30346] := B#16#0;
   STAT0[-30345] := B#16#0;
   STAT0[-30344] := B#16#0;
   STAT0[-30343] := B#16#0;
   STAT0[-30342] := B#16#0;
   STAT0[-30341] := B#16#0;
   STAT0[-30340] := B#16#0;
   STAT0[-30339] := B#16#0;
   STAT0[-30338] := B#16#0;
   STAT0[-30337] := B#16#0;
   STAT0[-30336] := B#16#0;
   STAT0[-30335] := B#16#0;
   STAT0[-30334] := B#16#0;
   STAT0[-30333] := B#16#0;
   STAT0[-30332] := B#16#0;
   STAT0[-30331] := B#16#0;
   STAT0[-30330] := B#16#0;
   STAT0[-30329] := B#16#0;
   STAT0[-30328] := B#16#0;
   STAT0[-30327] := B#16#0;
   STAT0[-30326] := B#16#0;
   STAT0[-30325] := B#16#0;
   STAT0[-30324] := B#16#0;
   STAT0[-30323] := B#16#0;
   STAT0[-30322] := B#16#0;
   STAT0[-30321] := B#16#0;
   STAT0[-30320] := B#16#0;
   STAT0[-30319] := B#16#0;
   STAT0[-30318] := B#16#0;
   STAT0[-30317] := B#16#0;
   STAT0[-30316] := B#16#0;
   STAT0[-30315] := B#16#0;
   STAT0[-30314] := B#16#0;
   STAT0[-30313] := B#16#0;
   STAT0[-30312] := B#16#0;
   STAT0[-30311] := B#16#0;
   STAT0[-30310] := B#16#0;
   STAT0[-30309] := B#16#0;
   STAT0[-30308] := B#16#0;
   STAT0[-30307] := B#16#0;
   STAT0[-30306] := B#16#0;
   STAT0[-30305] := B#16#0;
   STAT0[-30304] := B#16#0;
   STAT0[-30303] := B#16#0;
   STAT0[-30302] := B#16#0;
   STAT0[-30301] := B#16#0;
   STAT0[-30300] := B#16#0;
   STAT0[-30299] := B#16#0;
   STAT0[-30298] := B#16#0;
   STAT0[-30297] := B#16#0;
   STAT0[-30296] := B#16#0;
   STAT0[-30295] := B#16#0;
   STAT0[-30294] := B#16#0;
   STAT0[-30293] := B#16#0;
   STAT0[-30292] := B#16#0;
   STAT0[-30291] := B#16#0;
   STAT0[-30290] := B#16#0;
   STAT0[-30289] := B#16#0;
   STAT0[-30288] := B#16#0;
   STAT0[-30287] := B#16#0;
   STAT0[-30286] := B#16#0;
   STAT0[-30285] := B#16#0;
   STAT0[-30284] := B#16#0;
   STAT0[-30283] := B#16#0;
   STAT0[-30282] := B#16#0;
   STAT0[-30281] := B#16#0;
   STAT0[-30280] := B#16#0;
   STAT0[-30279] := B#16#0;
   STAT0[-30278] := B#16#0;
   STAT0[-30277] := B#16#0;
   STAT0[-30276] := B#16#0;
   STAT0[-30275] := B#16#0;
   STAT0[-30274] := B#16#0;
   STAT0[-30273] := B#16#0;
   STAT0[-30272] := B#16#0;
   STAT0[-30271] := B#16#0;
END_DATA_BLOCK

FUNCTION_BLOCK FB 402
TITLE =Operation Mode Select Program
AUTHOR : HMC
FAMILY : Mode
NAME : Mode
VERSION : 1.0


VAR_INPUT
  SSD_Manual : BOOL ;
  SSD_Auto : BOOL ;
  PB_Ready : BOOL ;
  PB_Auto_Run : BOOL ;
  PB_Remote_Ready : BOOL ;
  PB_Remote_Auto_Run : BOOL ;
  PB_Lamp_CHK : BOOL ;
  M_Air_Error : BOOL ;
  M_Water_Error : BOOL ;
  M_Total_Error : BOOL ;
  M_EStop : BOOL ;
  EXT_Ready : BOOL ;
  EXT_Auto : BOOL ;
  T_SemiAuto : TIME ;
  M_FLICK : BOOL ;
END_VAR
VAR_OUTPUT
  M_Ready_On : BOOL ;
  M_Auto_Mode : BOOL ;
  M_SemiAuto_Mode : BOOL ;
  M_Manual_Mode : BOOL ;
  M_Auto_Run : BOOL ;
  LP_Ready_On : BOOL ;
  LP_Auto_Run : BOOL ;
END_VAR
VAR
  AUTO_MODE_DELAY : SFB 4;
  SEMI_AUTO_DELAY : SFB 4;
  MANUAL_DELAY : SFB 4;
END_VAR
BEGIN
NETWORK
TITLE =Auto Mode Select Program
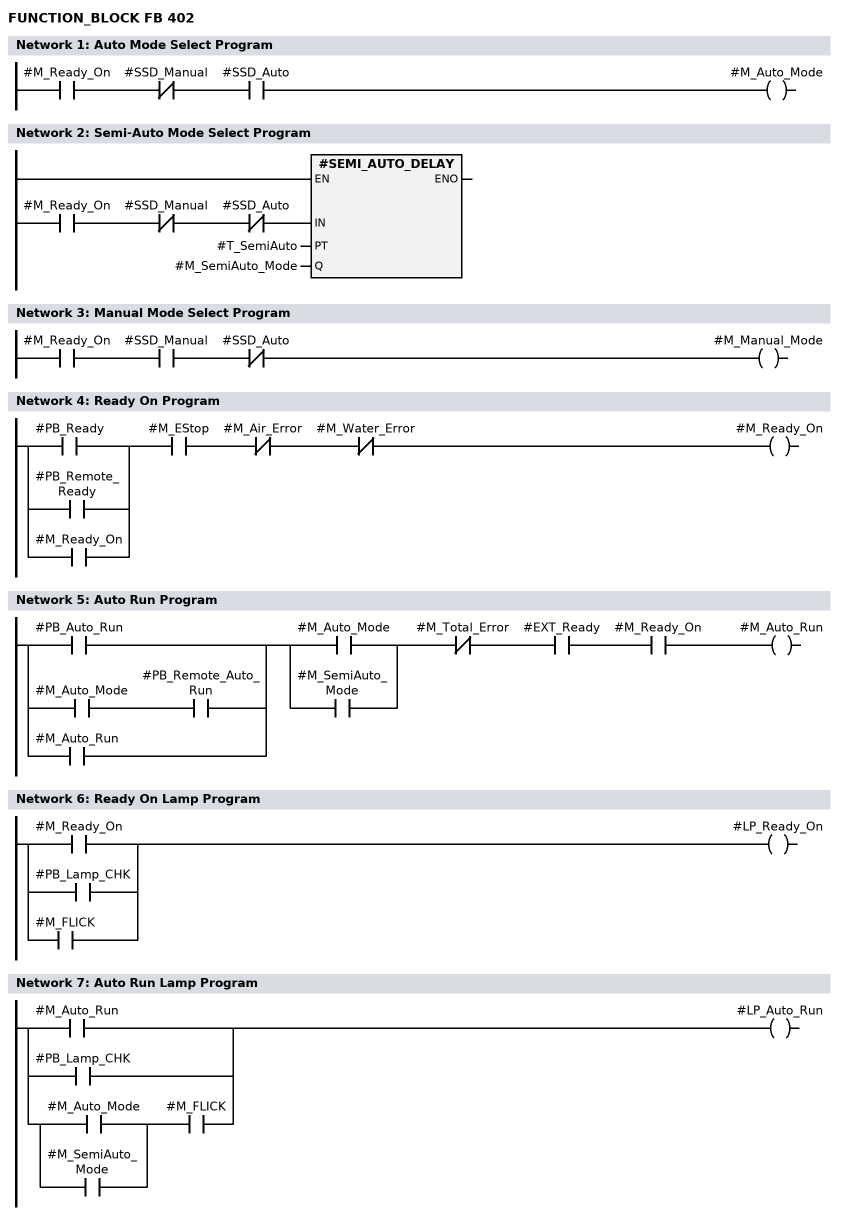

      A     #M_Ready_On;
      AN    #SSD_Manual;
      A     #SSD_Auto;
      =     #M_Auto_Mode;
NETWORK
TITLE =Semi-Auto Mode Select Program

      A     #M_Ready_On;
      AN    #SSD_Manual;
      AN    #SSD_Auto;
      =     L      0.0;
      BLD   103;
      CALL #SEMI_AUTO_DELAY (
           IN                       := L      0.0,
           PT                       := #T_SemiAuto,
           Q                        := #M_SemiAuto_Mode);

      NOP   0;
NETWORK
TITLE =Manual Mode Select Program

      A     #M_Ready_On;
      A     #SSD_Manual;
      AN    #SSD_Auto;
      =     #M_Manual_Mode;
NETWORK
TITLE =Ready On Program

      A(    ;
      O     #PB_Ready;
      O     #PB_Remote_Ready;
      O     #M_Ready_On;
      )     ;
      A     #M_EStop;
      AN    #M_Air_Error;
      AN    #M_Water_Error;
      =     #M_Ready_On;
NETWORK
TITLE =Auto Run Program

      A(    ;
      O     #PB_Auto_Run;
      O     ;
      A     #M_Auto_Mode;
      A     #PB_Remote_Auto_Run;
      O     #M_Auto_Run;
      )     ;
      A(    ;
      O     #M_Auto_Mode;
      O     #M_SemiAuto_Mode;
      )     ;
      AN    #M_Total_Error;
      A     #EXT_Ready;
      A     #M_Ready_On;
      =     #M_Auto_Run;
NETWORK
TITLE =Ready On Lamp Program

      O     #M_Ready_On;
      O     #PB_Lamp_CHK;
      O     #M_FLICK;
      =     #LP_Ready_On;
NETWORK
TITLE =Auto Run Lamp Program

      O     #M_Auto_Run;
      O     #PB_Lamp_CHK;
      O     ;
      A(    ;
      O     #M_Auto_Mode;
      O     #M_SemiAuto_Mode;
      )     ;
      A     #M_FLICK;
      =     #LP_Auto_Run;
END_FUNCTION_BLOCK

FUNCTION_BLOCK FB 424
TITLE =Sensor Error,Lamp Variables Program
AUTHOR : HMC
FAMILY : Common
NAME : Common
VERSION : 1.0


VAR_INPUT
  Enable_Aux : BOOL ;
  Adv_Amount : INT ;
  Ret_Amount : INT ;
  LS_Adv1 : BOOL ;
  LS_Ret1 : BOOL ;
  LS_Adv2 : BOOL ;
  LS_Ret2 : BOOL ;
  LS_Adv3 : BOOL ;
  LS_Ret3 : BOOL ;
  LS_Adv4 : BOOL ;
  LS_Ret4 : BOOL ;
  SOL_Adv : BOOL ;
  SOL_Ret : BOOL ;
  M_Ready : BOOL ;
  T_CHK1 : TIME ;
  T_CHK2 : TIME ;
  PB_Lamp_CHK : BOOL ;
  PB_Error_Rst : BOOL ;
  M_FLICK : BOOL ;
END_VAR
VAR_OUTPUT
  M_Adv_Err : BOOL ;
  M_Ret_Err : BOOL ;
  LP_Adv : BOOL ;
  LP_Ret : BOOL ;
  Visu_Adv : WORD ;
  Visu_Ret : WORD ;
END_VAR
VAR
  Error_T1 : SFB 4;
  Error_T2 : SFB 4;
  CHK_Aux1 : BOOL ;
  CHK_Aux2 : BOOL ;
  Error_T1_DN : BOOL ;
  Error_T2_DN : BOOL ;
  Adv_Memo : BOOL ;
  Visu_Adv_Arr : ARRAY  [0 .. 15 ] OF BOOL ;
  Visu_Ret_Arr : ARRAY  [0 .. 15 ] OF BOOL ;
  BLK_Move_Ret : INT ;
  Enable : BOOL ;
  Adv_End : BOOL ;
  Ret_End : BOOL ;
END_VAR
BEGIN
NETWORK
TITLE =
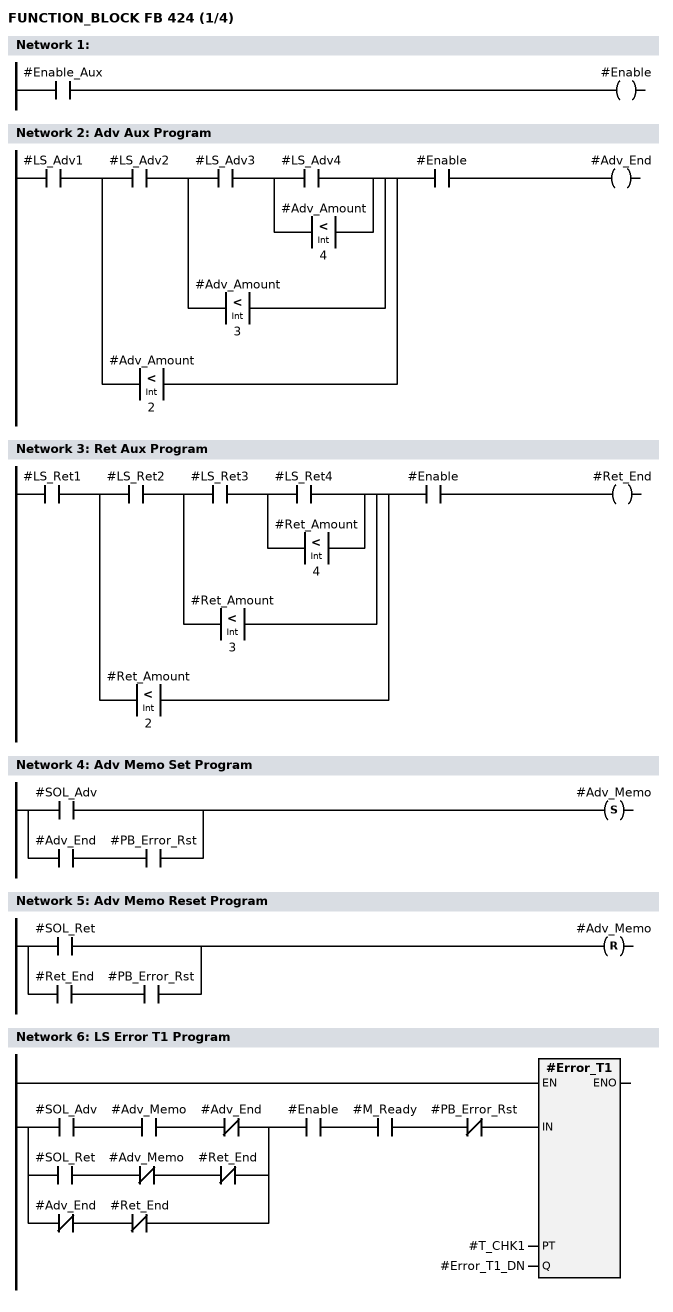

      A     #Enable_Aux;
      =     #Enable;
NETWORK
TITLE =Adv Aux Program

      A     #LS_Adv1;
      A(    ;
      A     #LS_Adv2;
      A(    ;
      A     #LS_Adv3;
      A(    ;
      O     #LS_Adv4;
      O(    ;
      L     #Adv_Amount;
      L     4;
      <I    ;
      )     ;
      )     ;
      O(    ;
      L     #Adv_Amount;
      L     3;
      <I    ;
      )     ;
      )     ;
      O(    ;
      L     #Adv_Amount;
      L     2;
      <I    ;
      )     ;
      )     ;
      A     #Enable;
      =     #Adv_End;
NETWORK
TITLE =Ret Aux Program

      A     #LS_Ret1;
      A(    ;
      A     #LS_Ret2;
      A(    ;
      A     #LS_Ret3;
      A(    ;
      O     #LS_Ret4;
      O(    ;
      L     #Ret_Amount;
      L     4;
      <I    ;
      )     ;
      )     ;
      O(    ;
      L     #Ret_Amount;
      L     3;
      <I    ;
      )     ;
      )     ;
      O(    ;
      L     #Ret_Amount;
      L     2;
      <I    ;
      )     ;
      )     ;
      A     #Enable;
      =     #Ret_End;
NETWORK
TITLE =Adv Memo Set Program

      O     #SOL_Adv;
      O     ;
      A     #Adv_End;
      A     #PB_Error_Rst;
      S     #Adv_Memo;
NETWORK
TITLE =Adv Memo Reset Program

      O     #SOL_Ret;
      O     ;
      A     #Ret_End;
      A     #PB_Error_Rst;
      R     #Adv_Memo;
NETWORK
TITLE =LS Error T1 Program

      A(    ;
      A     #SOL_Adv;
      A     #Adv_Memo;
      AN    #Adv_End;
      O     ;
      A     #SOL_Ret;
      AN    #Adv_Memo;
      AN    #Ret_End;
      O     ;
      AN    #Adv_End;
      AN    #Ret_End;
      )     ;
      A     #Enable;
      A     #M_Ready;
      AN    #PB_Error_Rst;
      =     L      0.0;
      BLD   103;
      CALL #Error_T1 (
           IN                       := L      0.0,
           PT                       := #T_CHK1,
           Q                        := #Error_T1_DN);

      NOP   0;
NETWORK
TITLE =Check Aux1 Program
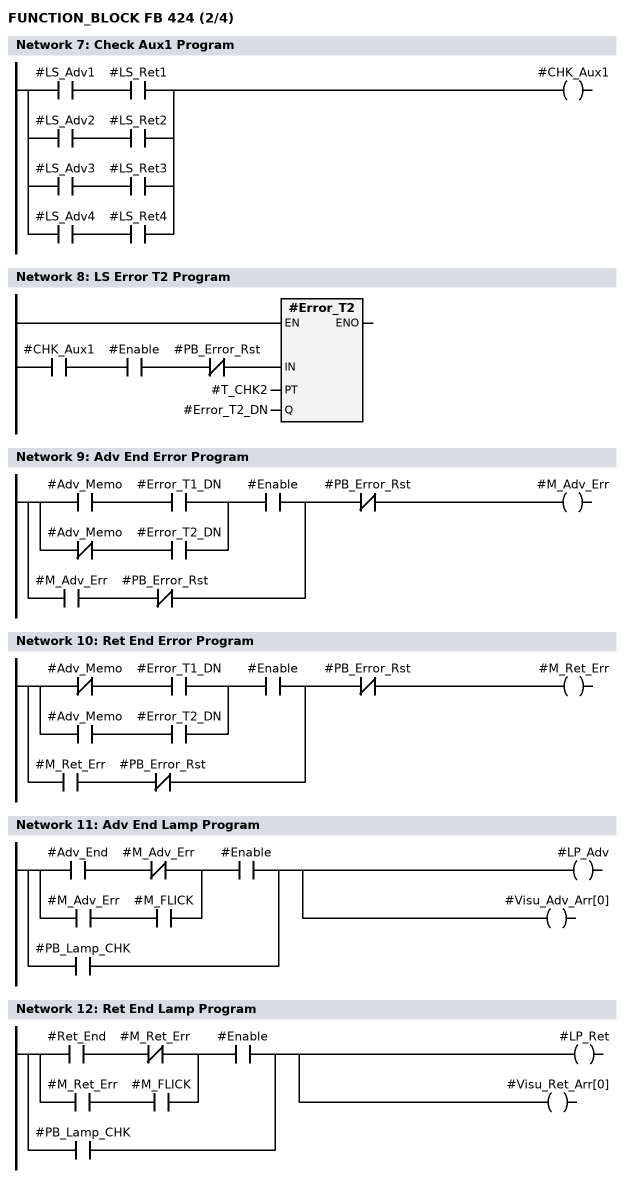

      A     #LS_Adv1;
      A     #LS_Ret1;
      O     ;
      A     #LS_Adv2;
      A     #LS_Ret2;
      O     ;
      A     #LS_Adv3;
      A     #LS_Ret3;
      O     ;
      A     #LS_Adv4;
      A     #LS_Ret4;
      =     #CHK_Aux1;
NETWORK
TITLE =LS Error T2 Program

      A     #CHK_Aux1;
      A     #Enable;
      AN    #PB_Error_Rst;
      =     L      0.0;
      BLD   103;
      CALL #Error_T2 (
           IN                       := L      0.0,
           PT                       := #T_CHK2,
           Q                        := #Error_T2_DN);

      NOP   0;
NETWORK
TITLE =Adv End Error Program

      A(    ;
      A(    ;
      A     #Adv_Memo;
      A     #Error_T1_DN;
      O     ;
      AN    #Adv_Memo;
      A     #Error_T2_DN;
      )     ;
      A     #Enable;
      O     ;
      A     #M_Adv_Err;
      AN    #PB_Error_Rst;
      )     ;
      AN    #PB_Error_Rst;
      =     #M_Adv_Err;
NETWORK
TITLE =Ret End Error Program

      A(    ;
      A(    ;
      AN    #Adv_Memo;
      A     #Error_T1_DN;
      O     ;
      A     #Adv_Memo;
      A     #Error_T2_DN;
      )     ;
      A     #Enable;
      O     ;
      A     #M_Ret_Err;
      AN    #PB_Error_Rst;
      )     ;
      AN    #PB_Error_Rst;
      =     #M_Ret_Err;
NETWORK
TITLE =Adv End Lamp Program

      A(    ;
      A     #Adv_End;
      AN    #M_Adv_Err;
      O     ;
      A     #M_Adv_Err;
      A     #M_FLICK;
      )     ;
      A     #Enable;
      O     #PB_Lamp_CHK;
      =     #LP_Adv;
      =     #Visu_Adv_Arr[0];
NETWORK
TITLE =Ret End Lamp Program

      A(    ;
      A     #Ret_End;
      AN    #M_Ret_Err;
      O     ;
      A     #M_Ret_Err;
      A     #M_FLICK;
      )     ;
      A     #Enable;
      O     #PB_Lamp_CHK;
      =     #LP_Ret;
      =     #Visu_Ret_Arr[0];
NETWORK
TITLE =Adv LS_1 Lamp Program
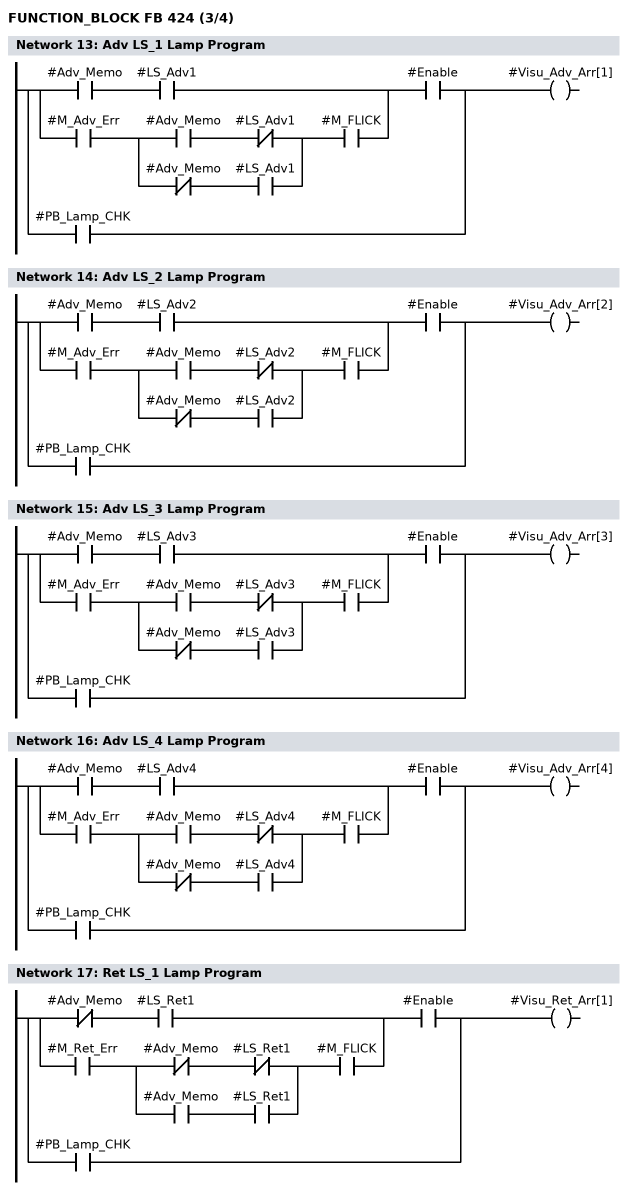

      A(    ;
      A     #Adv_Memo;
      A     #LS_Adv1;
      O     ;
      A     #M_Adv_Err;
      A(    ;
      A     #Adv_Memo;
      AN    #LS_Adv1;
      O     ;
      AN    #Adv_Memo;
      A     #LS_Adv1;
      )     ;
      A     #M_FLICK;
      )     ;
      A     #Enable;
      O     #PB_Lamp_CHK;
      =     #Visu_Adv_Arr[1];
NETWORK
TITLE =Adv LS_2 Lamp Program
//
//
      A(    ;
      A     #Adv_Memo;
      A     #LS_Adv2;
      O     ;
      A     #M_Adv_Err;
      A(    ;
      A     #Adv_Memo;
      AN    #LS_Adv2;
      O     ;
      AN    #Adv_Memo;
      A     #LS_Adv2;
      )     ;
      A     #M_FLICK;
      )     ;
      A     #Enable;
      O     #PB_Lamp_CHK;
      =     #Visu_Adv_Arr[2];
NETWORK
TITLE =Adv LS_3 Lamp Program
//
//
      A(    ;
      A     #Adv_Memo;
      A     #LS_Adv3;
      O     ;
      A     #M_Adv_Err;
      A(    ;
      A     #Adv_Memo;
      AN    #LS_Adv3;
      O     ;
      AN    #Adv_Memo;
      A     #LS_Adv3;
      )     ;
      A     #M_FLICK;
      )     ;
      A     #Enable;
      O     #PB_Lamp_CHK;
      =     #Visu_Adv_Arr[3];
NETWORK
TITLE =Adv LS_4 Lamp Program
//
//
      A(    ;
      A     #Adv_Memo;
      A     #LS_Adv4;
      O     ;
      A     #M_Adv_Err;
      A(    ;
      A     #Adv_Memo;
      AN    #LS_Adv4;
      O     ;
      AN    #Adv_Memo;
      A     #LS_Adv4;
      )     ;
      A     #M_FLICK;
      )     ;
      A     #Enable;
      O     #PB_Lamp_CHK;
      =     #Visu_Adv_Arr[4];
NETWORK
TITLE =Ret LS_1 Lamp Program
//
//
      A(    ;
      AN    #Adv_Memo;
      A     #LS_Ret1;
      O     ;
      A     #M_Ret_Err;
      A(    ;
      AN    #Adv_Memo;
      AN    #LS_Ret1;
      O     ;
      A     #Adv_Memo;
      A     #LS_Ret1;
      )     ;
      A     #M_FLICK;
      )     ;
      A     #Enable;
      O     #PB_Lamp_CHK;
      =     #Visu_Ret_Arr[1];
NETWORK
TITLE =Ret LS_2 Lamp Program
//
//
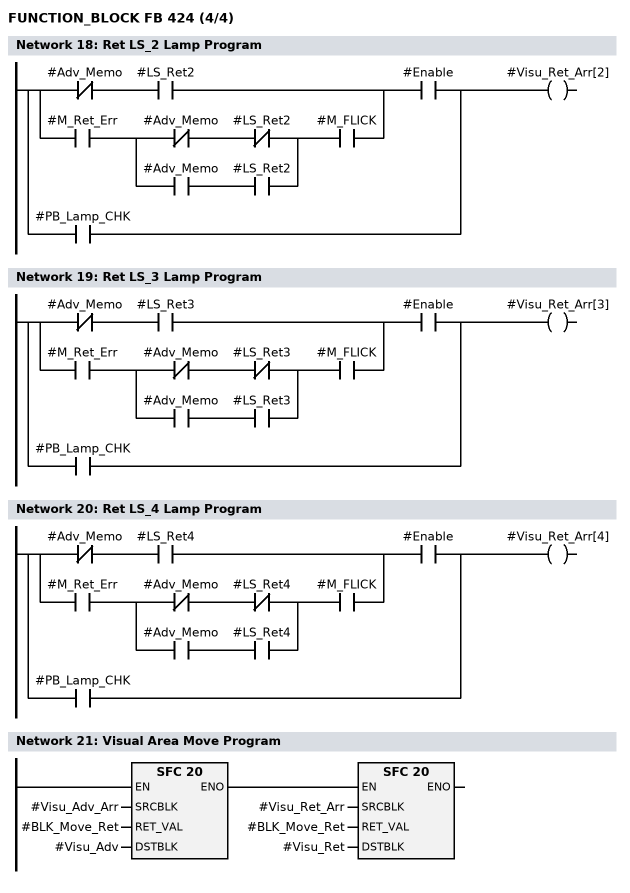
      A(    ;
      AN    #Adv_Memo;
      A     #LS_Ret2;
      O     ;
      A     #M_Ret_Err;
      A(    ;
      AN    #Adv_Memo;
      AN    #LS_Ret2;
      O     ;
      A     #Adv_Memo;
      A     #LS_Ret2;
      )     ;
      A     #M_FLICK;
      )     ;
      A     #Enable;
      O     #PB_Lamp_CHK;
      =     #Visu_Ret_Arr[2];
NETWORK
TITLE =Ret LS_3 Lamp Program
//
//
      A(    ;
      AN    #Adv_Memo;
      A     #LS_Ret3;
      O     ;
      A     #M_Ret_Err;
      A(    ;
      AN    #Adv_Memo;
      AN    #LS_Ret3;
      O     ;
      A     #Adv_Memo;
      A     #LS_Ret3;
      )     ;
      A     #M_FLICK;
      )     ;
      A     #Enable;
      O     #PB_Lamp_CHK;
      =     #Visu_Ret_Arr[3];
NETWORK
TITLE =Ret LS_4 Lamp Program
//
//
      A(    ;
      AN    #Adv_Memo;
      A     #LS_Ret4;
      O     ;
      A     #M_Ret_Err;
      A(    ;
      AN    #Adv_Memo;
      AN    #LS_Ret4;
      O     ;
      A     #Adv_Memo;
      A     #LS_Ret4;
      )     ;
      A     #M_FLICK;
      )     ;
      A     #Enable;
      O     #PB_Lamp_CHK;
      =     #Visu_Ret_Arr[4];
NETWORK
TITLE =Visual Area Move Program

      A(    ;
      CALL SFC   20 (
           SRCBLK                   := #Visu_Adv_Arr,
           RET_VAL                  := #BLK_Move_Ret,
           DSTBLK                   := #Visu_Adv);
      A     BR;
      )     ;
      JNB   _001;
      CALL SFC   20 (
           SRCBLK                   := #Visu_Ret_Arr,
           RET_VAL                  := #BLK_Move_Ret,
           DSTBLK                   := #Visu_Ret);
_001: NOP   0;
END_FUNCTION_BLOCK

FUNCTION_BLOCK FB 426
TITLE =Sensor Error,Lamp Variables Program
AUTHOR : HMC
FAMILY : Common
NAME : Common
VERSION : 1.0


VAR_INPUT
  Enable_Aux : BOOL ;
  Adv_Amount : INT ;
  Ret_Amount : INT ;
  LS_Adv1 : BOOL ;
  LS_Ret1 : BOOL ;
  LS_Adv2 : BOOL ;
  LS_Ret2 : BOOL ;
  LS_Adv3 : BOOL ;
  LS_Ret3 : BOOL ;
  LS_Adv4 : BOOL ;
  LS_Ret4 : BOOL ;
  LS_Adv5 : BOOL ;
  LS_Ret5 : BOOL ;
  LS_Adv6 : BOOL ;
  LS_Ret6 : BOOL ;
  LS_Adv7 : BOOL ;
  LS_Ret7 : BOOL ;
  LS_Adv8 : BOOL ;
  LS_Ret8 : BOOL ;
  SOL_Adv : BOOL ;
  SOL_Ret : BOOL ;
  M_Ready : BOOL ;
  T_CHK1 : TIME ;
  T_CHK2 : TIME ;
  PB_Lamp_CHK : BOOL ;
  PB_Error_Rst : BOOL ;
  M_FLICK : BOOL ;
END_VAR
VAR_OUTPUT
  M_Adv_Err : BOOL ;
  M_Ret_Err : BOOL ;
  LP_Adv : BOOL ;
  LP_Ret : BOOL ;
  Visu_Adv : WORD ;
  Visu_Ret : WORD ;
END_VAR
VAR
  Error_T1 : SFB 4;
  Error_T2 : SFB 4;
  Adv_End_Aux : BOOL ;
  Ret_End_Aux : BOOL ;
  CHK_Aux1 : BOOL ;
  CHK_Aux2 : BOOL ;
  Error_T1_DN : BOOL ;
  Error_T2_DN : BOOL ;
  Adv_Memo : BOOL ;
  Visu_Adv_Arr : ARRAY  [0 .. 15 ] OF BOOL ;
  Visu_Ret_Arr : ARRAY  [0 .. 15 ] OF BOOL ;
  BLK_Move_Ret : INT ;
  Enable : BOOL ;
  Adv_End : BOOL ;
  Ret_End : BOOL ;
END_VAR
BEGIN
NETWORK
TITLE =
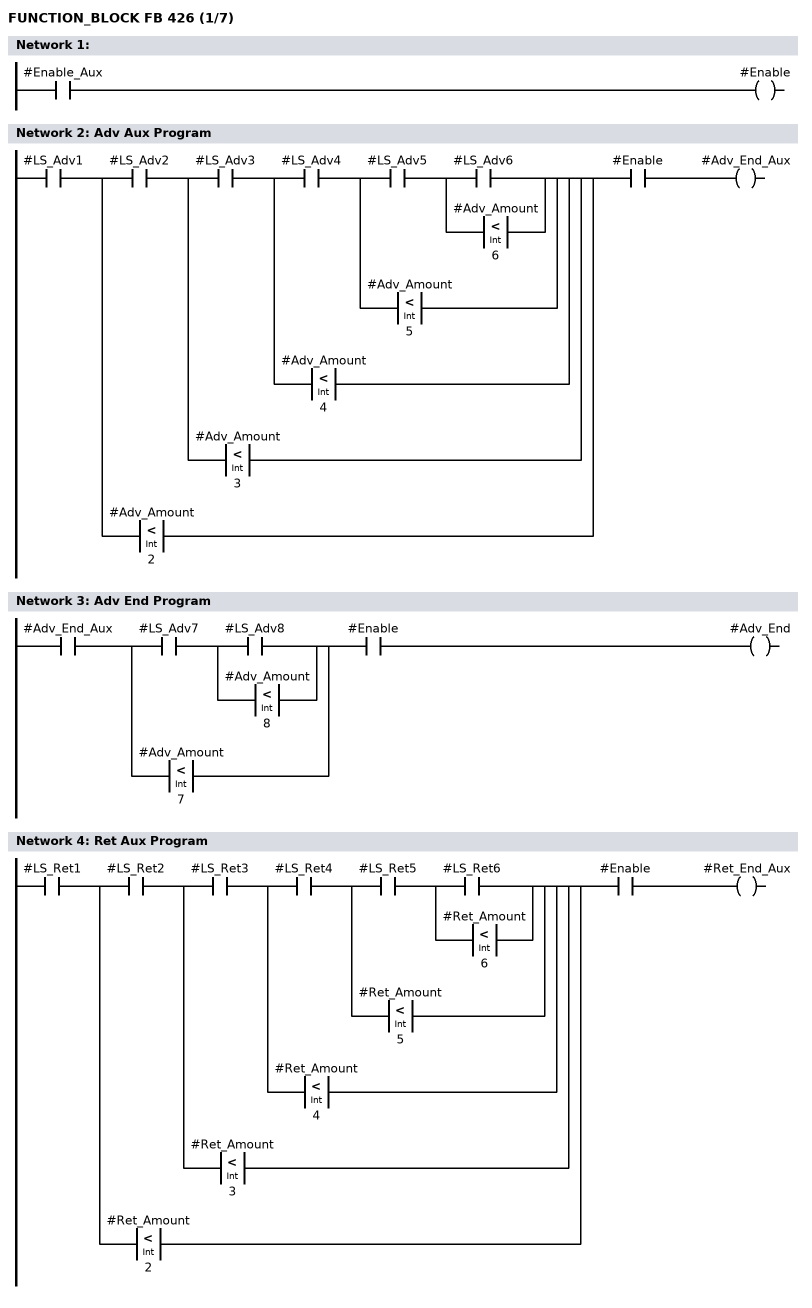

      A     #Enable_Aux;
      =     #Enable;
NETWORK
TITLE =Adv Aux Program

      A     #LS_Adv1;
      A(    ;
      A     #LS_Adv2;
      A(    ;
      A     #LS_Adv3;
      A(    ;
      A     #LS_Adv4;
      A(    ;
      A     #LS_Adv5;
      A(    ;
      O     #LS_Adv6;
      O(    ;
      L     #Adv_Amount;
      L     6;
      <I    ;
      )     ;
      )     ;
      O(    ;
      L     #Adv_Amount;
      L     5;
      <I    ;
      )     ;
      )     ;
      O(    ;
      L     #Adv_Amount;
      L     4;
      <I    ;
      )     ;
      )     ;
      O(    ;
      L     #Adv_Amount;
      L     3;
      <I    ;
      )     ;
      )     ;
      O(    ;
      L     #Adv_Amount;
      L     2;
      <I    ;
      )     ;
      )     ;
      A     #Enable;
      =     #Adv_End_Aux;
NETWORK
TITLE =Adv End Program

      A     #Adv_End_Aux;
      A(    ;
      A     #LS_Adv7;
      A(    ;
      O     #LS_Adv8;
      O(    ;
      L     #Adv_Amount;
      L     8;
      <I    ;
      )     ;
      )     ;
      O(    ;
      L     #Adv_Amount;
      L     7;
      <I    ;
      )     ;
      )     ;
      A     #Enable;
      =     #Adv_End;
NETWORK
TITLE =Ret Aux Program

      A     #LS_Ret1;
      A(    ;
      A     #LS_Ret2;
      A(    ;
      A     #LS_Ret3;
      A(    ;
      A     #LS_Ret4;
      A(    ;
      A     #LS_Ret5;
      A(    ;
      O     #LS_Ret6;
      O(    ;
      L     #Ret_Amount;
      L     6;
      <I    ;
      )     ;
      )     ;
      O(    ;
      L     #Ret_Amount;
      L     5;
      <I    ;
      )     ;
      )     ;
      O(    ;
      L     #Ret_Amount;
      L     4;
      <I    ;
      )     ;
      )     ;
      O(    ;
      L     #Ret_Amount;
      L     3;
      <I    ;
      )     ;
      )     ;
      O(    ;
      L     #Ret_Amount;
      L     2;
      <I    ;
      )     ;
      )     ;
      A     #Enable;
      =     #Ret_End_Aux;
NETWORK
TITLE =Ret End Program
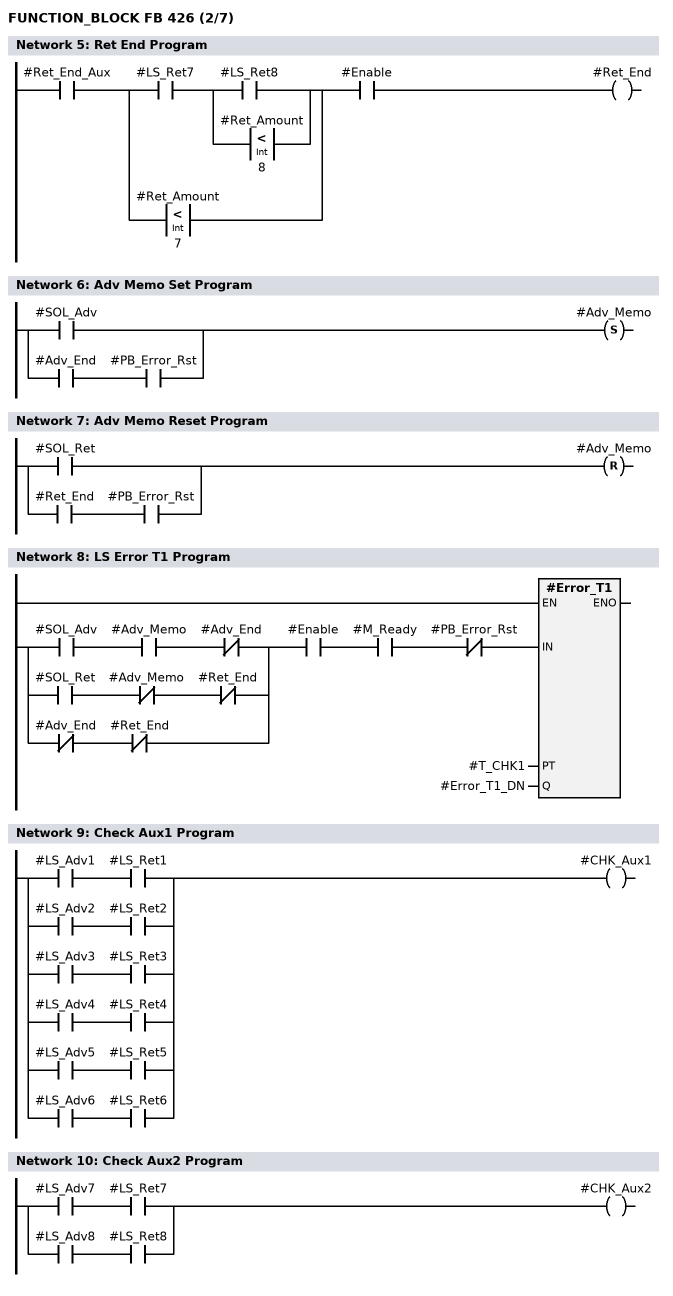

      A     #Ret_End_Aux;
      A(    ;
      A     #LS_Ret7;
      A(    ;
      O     #LS_Ret8;
      O(    ;
      L     #Ret_Amount;
      L     8;
      <I    ;
      )     ;
      )     ;
      O(    ;
      L     #Ret_Amount;
      L     7;
      <I    ;
      )     ;
      )     ;
      A     #Enable;
      =     #Ret_End;
NETWORK
TITLE =Adv Memo Set Program

      O     #SOL_Adv;
      O     ;
      A     #Adv_End;
      A     #PB_Error_Rst;
      S     #Adv_Memo;
NETWORK
TITLE =Adv Memo Reset Program

      O     #SOL_Ret;
      O     ;
      A     #Ret_End;
      A     #PB_Error_Rst;
      R     #Adv_Memo;
NETWORK
TITLE =LS Error T1 Program

      A(    ;
      A     #SOL_Adv;
      A     #Adv_Memo;
      AN    #Adv_End;
      O     ;
      A     #SOL_Ret;
      AN    #Adv_Memo;
      AN    #Ret_End;
      O     ;
      AN    #Adv_End;
      AN    #Ret_End;
      )     ;
      A     #Enable;
      A     #M_Ready;
      AN    #PB_Error_Rst;
      =     L      0.0;
      BLD   103;
      CALL #Error_T1 (
           IN                       := L      0.0,
           PT                       := #T_CHK1,
           Q                        := #Error_T1_DN);

      NOP   0;
NETWORK
TITLE =Check Aux1 Program

      A     #LS_Adv1;
      A     #LS_Ret1;
      O     ;
      A     #LS_Adv2;
      A     #LS_Ret2;
      O     ;
      A     #LS_Adv3;
      A     #LS_Ret3;
      O     ;
      A     #LS_Adv4;
      A     #LS_Ret4;
      O     ;
      A     #LS_Adv5;
      A     #LS_Ret5;
      O     ;
      A     #LS_Adv6;
      A     #LS_Ret6;
      =     #CHK_Aux1;
NETWORK
TITLE =Check Aux2 Program

      A     #LS_Adv7;
      A     #LS_Ret7;
      O     ;
      A     #LS_Adv8;
      A     #LS_Ret8;
      =     #CHK_Aux2;
NETWORK
TITLE =LS Error T2 Program
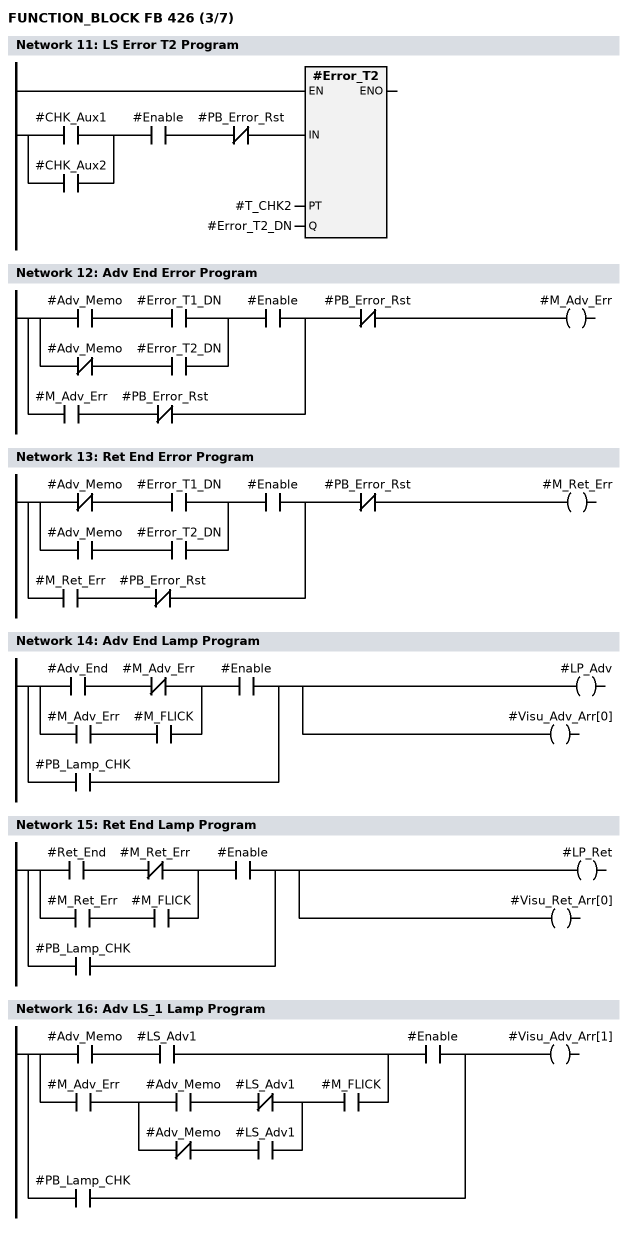

      A(    ;
      O     #CHK_Aux1;
      O     #CHK_Aux2;
      )     ;
      A     #Enable;
      AN    #PB_Error_Rst;
      =     L      0.0;
      BLD   103;
      CALL #Error_T2 (
           IN                       := L      0.0,
           PT                       := #T_CHK2,
           Q                        := #Error_T2_DN);

      NOP   0;
NETWORK
TITLE =Adv End Error Program

      A(    ;
      A(    ;
      A     #Adv_Memo;
      A     #Error_T1_DN;
      O     ;
      AN    #Adv_Memo;
      A     #Error_T2_DN;
      )     ;
      A     #Enable;
      O     ;
      A     #M_Adv_Err;
      AN    #PB_Error_Rst;
      )     ;
      AN    #PB_Error_Rst;
      =     #M_Adv_Err;
NETWORK
TITLE =Ret End Error Program

      A(    ;
      A(    ;
      AN    #Adv_Memo;
      A     #Error_T1_DN;
      O     ;
      A     #Adv_Memo;
      A     #Error_T2_DN;
      )     ;
      A     #Enable;
      O     ;
      A     #M_Ret_Err;
      AN    #PB_Error_Rst;
      )     ;
      AN    #PB_Error_Rst;
      =     #M_Ret_Err;
NETWORK
TITLE =Adv End Lamp Program

      A(    ;
      A     #Adv_End;
      AN    #M_Adv_Err;
      O     ;
      A     #M_Adv_Err;
      A     #M_FLICK;
      )     ;
      A     #Enable;
      O     #PB_Lamp_CHK;
      =     #LP_Adv;
      =     #Visu_Adv_Arr[0];
NETWORK
TITLE =Ret End Lamp Program

      A(    ;
      A     #Ret_End;
      AN    #M_Ret_Err;
      O     ;
      A     #M_Ret_Err;
      A     #M_FLICK;
      )     ;
      A     #Enable;
      O     #PB_Lamp_CHK;
      =     #LP_Ret;
      =     #Visu_Ret_Arr[0];
NETWORK
TITLE =Adv LS_1 Lamp Program

      A(    ;
      A     #Adv_Memo;
      A     #LS_Adv1;
      O     ;
      A     #M_Adv_Err;
      A(    ;
      A     #Adv_Memo;
      AN    #LS_Adv1;
      O     ;
      AN    #Adv_Memo;
      A     #LS_Adv1;
      )     ;
      A     #M_FLICK;
      )     ;
      A     #Enable;
      O     #PB_Lamp_CHK;
      =     #Visu_Adv_Arr[1];
NETWORK
TITLE =Adv LS_2 Lamp Program
//
//
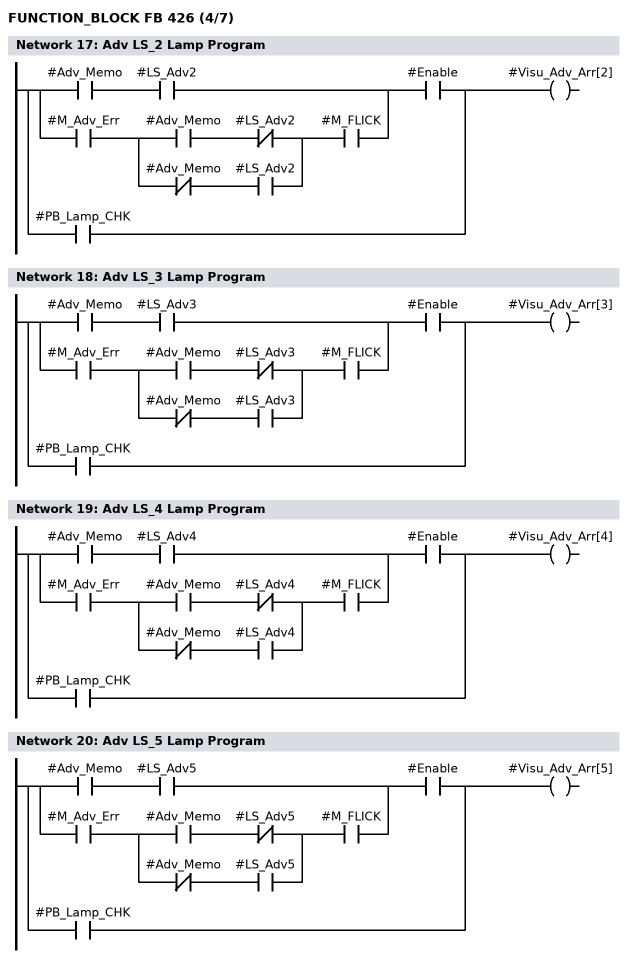
      A(    ;
      A     #Adv_Memo;
      A     #LS_Adv2;
      O     ;
      A     #M_Adv_Err;
      A(    ;
      A     #Adv_Memo;
      AN    #LS_Adv2;
      O     ;
      AN    #Adv_Memo;
      A     #LS_Adv2;
      )     ;
      A     #M_FLICK;
      )     ;
      A     #Enable;
      O     #PB_Lamp_CHK;
      =     #Visu_Adv_Arr[2];
NETWORK
TITLE =Adv LS_3 Lamp Program
//
//
      A(    ;
      A     #Adv_Memo;
      A     #LS_Adv3;
      O     ;
      A     #M_Adv_Err;
      A(    ;
      A     #Adv_Memo;
      AN    #LS_Adv3;
      O     ;
      AN    #Adv_Memo;
      A     #LS_Adv3;
      )     ;
      A     #M_FLICK;
      )     ;
      A     #Enable;
      O     #PB_Lamp_CHK;
      =     #Visu_Adv_Arr[3];
NETWORK
TITLE =Adv LS_4 Lamp Program
//
//
      A(    ;
      A     #Adv_Memo;
      A     #LS_Adv4;
      O     ;
      A     #M_Adv_Err;
      A(    ;
      A     #Adv_Memo;
      AN    #LS_Adv4;
      O     ;
      AN    #Adv_Memo;
      A     #LS_Adv4;
      )     ;
      A     #M_FLICK;
      )     ;
      A     #Enable;
      O     #PB_Lamp_CHK;
      =     #Visu_Adv_Arr[4];
NETWORK
TITLE =Adv LS_5 Lamp Program
//
//
      A(    ;
      A     #Adv_Memo;
      A     #LS_Adv5;
      O     ;
      A     #M_Adv_Err;
      A(    ;
      A     #Adv_Memo;
      AN    #LS_Adv5;
      O     ;
      AN    #Adv_Memo;
      A     #LS_Adv5;
      )     ;
      A     #M_FLICK;
      )     ;
      A     #Enable;
      O     #PB_Lamp_CHK;
      =     #Visu_Adv_Arr[5];
NETWORK
TITLE =Adv LS_6 Lamp Program
//
//
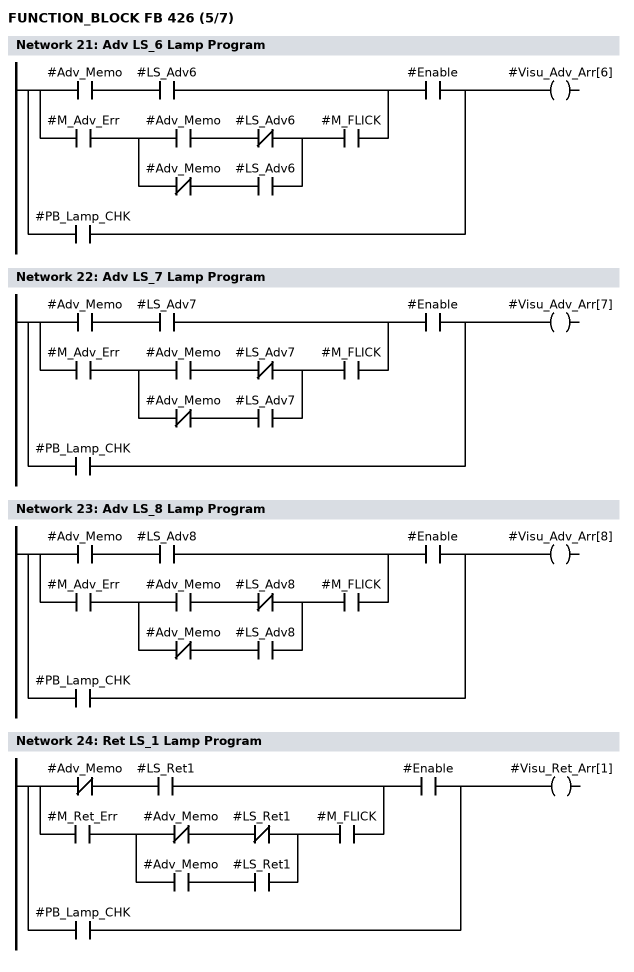
      A(    ;
      A     #Adv_Memo;
      A     #LS_Adv6;
      O     ;
      A     #M_Adv_Err;
      A(    ;
      A     #Adv_Memo;
      AN    #LS_Adv6;
      O     ;
      AN    #Adv_Memo;
      A     #LS_Adv6;
      )     ;
      A     #M_FLICK;
      )     ;
      A     #Enable;
      O     #PB_Lamp_CHK;
      =     #Visu_Adv_Arr[6];
NETWORK
TITLE =Adv LS_7 Lamp Program
//
//
      A(    ;
      A     #Adv_Memo;
      A     #LS_Adv7;
      O     ;
      A     #M_Adv_Err;
      A(    ;
      A     #Adv_Memo;
      AN    #LS_Adv7;
      O     ;
      AN    #Adv_Memo;
      A     #LS_Adv7;
      )     ;
      A     #M_FLICK;
      )     ;
      A     #Enable;
      O     #PB_Lamp_CHK;
      =     #Visu_Adv_Arr[7];
NETWORK
TITLE =Adv LS_8 Lamp Program
//
//
      A(    ;
      A     #Adv_Memo;
      A     #LS_Adv8;
      O     ;
      A     #M_Adv_Err;
      A(    ;
      A     #Adv_Memo;
      AN    #LS_Adv8;
      O     ;
      AN    #Adv_Memo;
      A     #LS_Adv8;
      )     ;
      A     #M_FLICK;
      )     ;
      A     #Enable;
      O     #PB_Lamp_CHK;
      =     #Visu_Adv_Arr[8];
NETWORK
TITLE =Ret LS_1 Lamp Program
//
//
      A(    ;
      AN    #Adv_Memo;
      A     #LS_Ret1;
      O     ;
      A     #M_Ret_Err;
      A(    ;
      AN    #Adv_Memo;
      AN    #LS_Ret1;
      O     ;
      A     #Adv_Memo;
      A     #LS_Ret1;
      )     ;
      A     #M_FLICK;
      )     ;
      A     #Enable;
      O     #PB_Lamp_CHK;
      =     #Visu_Ret_Arr[1];
NETWORK
TITLE =Ret LS_2 Lamp Program
//
//
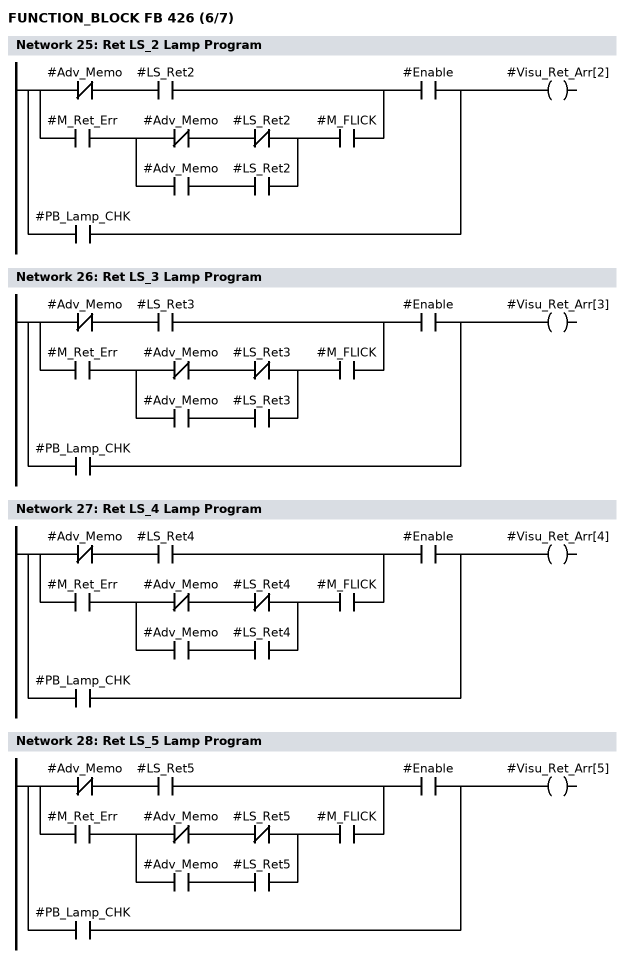
      A(    ;
      AN    #Adv_Memo;
      A     #LS_Ret2;
      O     ;
      A     #M_Ret_Err;
      A(    ;
      AN    #Adv_Memo;
      AN    #LS_Ret2;
      O     ;
      A     #Adv_Memo;
      A     #LS_Ret2;
      )     ;
      A     #M_FLICK;
      )     ;
      A     #Enable;
      O     #PB_Lamp_CHK;
      =     #Visu_Ret_Arr[2];
NETWORK
TITLE =Ret LS_3 Lamp Program
//
//
      A(    ;
      AN    #Adv_Memo;
      A     #LS_Ret3;
      O     ;
      A     #M_Ret_Err;
      A(    ;
      AN    #Adv_Memo;
      AN    #LS_Ret3;
      O     ;
      A     #Adv_Memo;
      A     #LS_Ret3;
      )     ;
      A     #M_FLICK;
      )     ;
      A     #Enable;
      O     #PB_Lamp_CHK;
      =     #Visu_Ret_Arr[3];
NETWORK
TITLE =Ret LS_4 Lamp Program
//
//
      A(    ;
      AN    #Adv_Memo;
      A     #LS_Ret4;
      O     ;
      A     #M_Ret_Err;
      A(    ;
      AN    #Adv_Memo;
      AN    #LS_Ret4;
      O     ;
      A     #Adv_Memo;
      A     #LS_Ret4;
      )     ;
      A     #M_FLICK;
      )     ;
      A     #Enable;
      O     #PB_Lamp_CHK;
      =     #Visu_Ret_Arr[4];
NETWORK
TITLE =Ret LS_5 Lamp Program
//
//
      A(    ;
      AN    #Adv_Memo;
      A     #LS_Ret5;
      O     ;
      A     #M_Ret_Err;
      A(    ;
      AN    #Adv_Memo;
      AN    #LS_Ret5;
      O     ;
      A     #Adv_Memo;
      A     #LS_Ret5;
      )     ;
      A     #M_FLICK;
      )     ;
      A     #Enable;
      O     #PB_Lamp_CHK;
      =     #Visu_Ret_Arr[5];
NETWORK
TITLE =Ret LS_6 Lamp Program
//
//
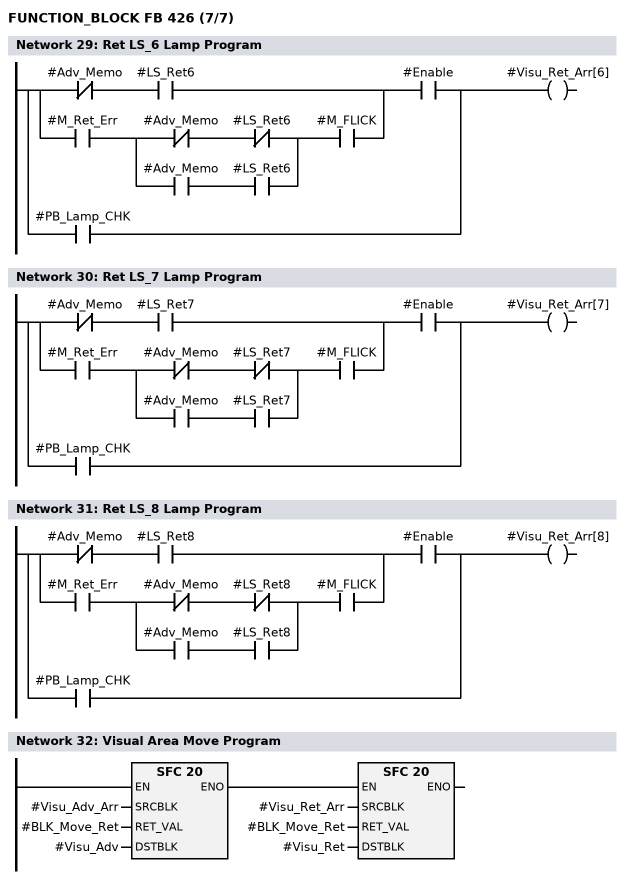
      A(    ;
      AN    #Adv_Memo;
      A     #LS_Ret6;
      O     ;
      A     #M_Ret_Err;
      A(    ;
      AN    #Adv_Memo;
      AN    #LS_Ret6;
      O     ;
      A     #Adv_Memo;
      A     #LS_Ret6;
      )     ;
      A     #M_FLICK;
      )     ;
      A     #Enable;
      O     #PB_Lamp_CHK;
      =     #Visu_Ret_Arr[6];
NETWORK
TITLE =Ret LS_7 Lamp Program
//
//
      A(    ;
      AN    #Adv_Memo;
      A     #LS_Ret7;
      O     ;
      A     #M_Ret_Err;
      A(    ;
      AN    #Adv_Memo;
      AN    #LS_Ret7;
      O     ;
      A     #Adv_Memo;
      A     #LS_Ret7;
      )     ;
      A     #M_FLICK;
      )     ;
      A     #Enable;
      O     #PB_Lamp_CHK;
      =     #Visu_Ret_Arr[7];
NETWORK
TITLE =Ret LS_8 Lamp Program
//
//
      A(    ;
      AN    #Adv_Memo;
      A     #LS_Ret8;
      O     ;
      A     #M_Ret_Err;
      A(    ;
      AN    #Adv_Memo;
      AN    #LS_Ret8;
      O     ;
      A     #Adv_Memo;
      A     #LS_Ret8;
      )     ;
      A     #M_FLICK;
      )     ;
      A     #Enable;
      O     #PB_Lamp_CHK;
      =     #Visu_Ret_Arr[8];
NETWORK
TITLE =Visual Area Move Program

      A(    ;
      CALL SFC   20 (
           SRCBLK                   := #Visu_Adv_Arr,
           RET_VAL                  := #BLK_Move_Ret,
           DSTBLK                   := #Visu_Adv);
      A     BR;
      )     ;
      JNB   _001;
      CALL SFC   20 (
           SRCBLK                   := #Visu_Ret_Arr,
           RET_VAL                  := #BLK_Move_Ret,
           DSTBLK                   := #Visu_Ret);
_001: NOP   0;
END_FUNCTION_BLOCK

FUNCTION FC 98 : VOID
TITLE =
VERSION : 0.1


VAR_TEMP
  SFC20_RET_VAL : INT ;
  RECV1_LEN : WORD ;
  SEND1_LEN : WORD ;
  RECV2_LEN : WORD ;
  SEND2_LEN : WORD ;
  RECV3_LEN : WORD ;
  SEND3_LEN : WORD ;
  RECV4_LEN : WORD ;
  SEND4_LEN : WORD ;
  RECV5_LEN : WORD ;
  SEND5_LEN : WORD ;
END_VAR
BEGIN
NETWORK
TITLE =
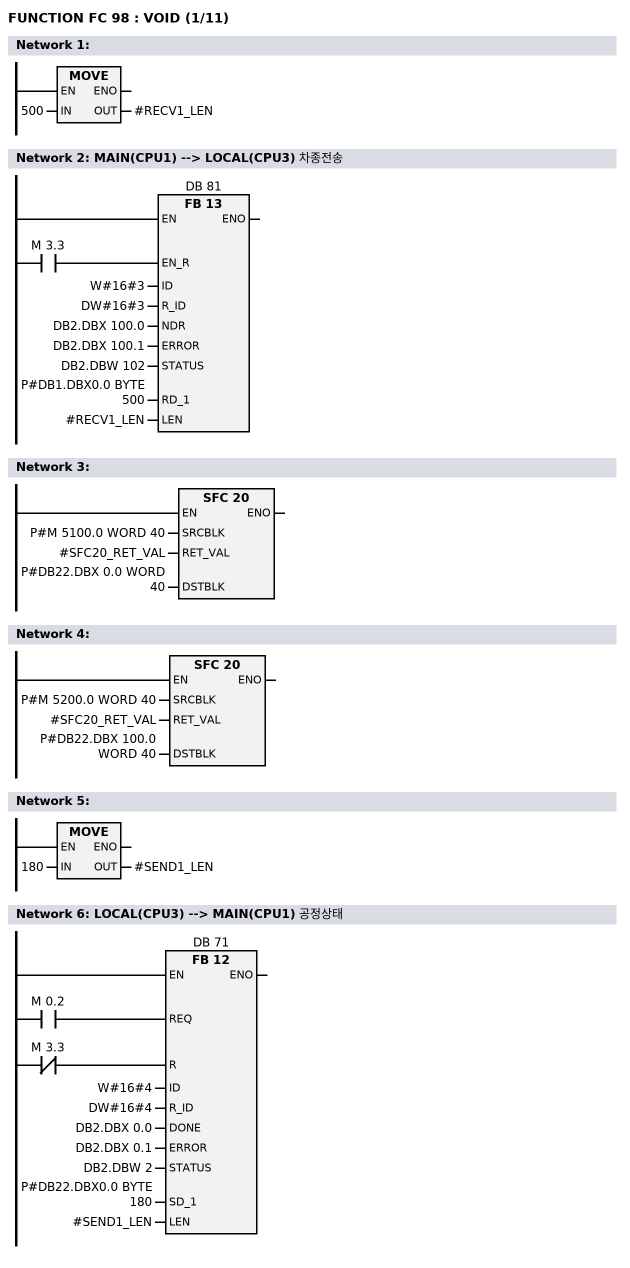

      L     500;
      T     #RECV1_LEN;
      NOP   0;
NETWORK
TITLE =MAIN(CPU1) --> LOCAL(CPU3) 차종전송

      A     M      3.3;
      =     L     22.0;
      BLD   103;
      CALL FB    13 , DB    81 (
           EN_R                     := L     22.0,
           ID                       := W#16#3,
           R_ID                     := DW#16#3,
           NDR                      := DB2.DBX  100.0,
           ERROR                    := DB2.DBX  100.1,
           STATUS                   := DB2.DBW  102,
           RD_1                     := P#DB1.DBX0.0 BYTE 500,
           LEN                      := #RECV1_LEN);
      NOP   0;
NETWORK
TITLE =

      CALL SFC   20 (
           SRCBLK                   := P#M 5100.0 WORD 40,
           RET_VAL                  := #SFC20_RET_VAL,
           DSTBLK                   := P#DB22.DBX 0.0 WORD 40);
      NOP   0;
NETWORK
TITLE =

      CALL SFC   20 (
           SRCBLK                   := P#M 5200.0 WORD 40,
           RET_VAL                  := #SFC20_RET_VAL,
           DSTBLK                   := P#DB22.DBX 100.0 WORD 40);
      NOP   0;
NETWORK
TITLE =

      L     180;
      T     #SEND1_LEN;
      NOP   0;
NETWORK
TITLE =LOCAL(CPU3) --> MAIN(CPU1) 공정상태
//
//
      A     M      0.2;
      =     L     22.0;
      BLD   103;
      AN    M      3.3;
      =     L     22.1;
      BLD   103;
      CALL FB    12 , DB    71 (
           REQ                      := L     22.0,
           R                        := L     22.1,
           ID                       := W#16#4,
           R_ID                     := DW#16#4,
           DONE                     := DB2.DBX    0.0,
           ERROR                    := DB2.DBX    0.1,
           STATUS                   := DB2.DBW    2,
           SD_1                     := P#DB22.DBX0.0 BYTE 180,
           LEN                      := #SEND1_LEN);
      NOP   0;
NETWORK
TITLE =
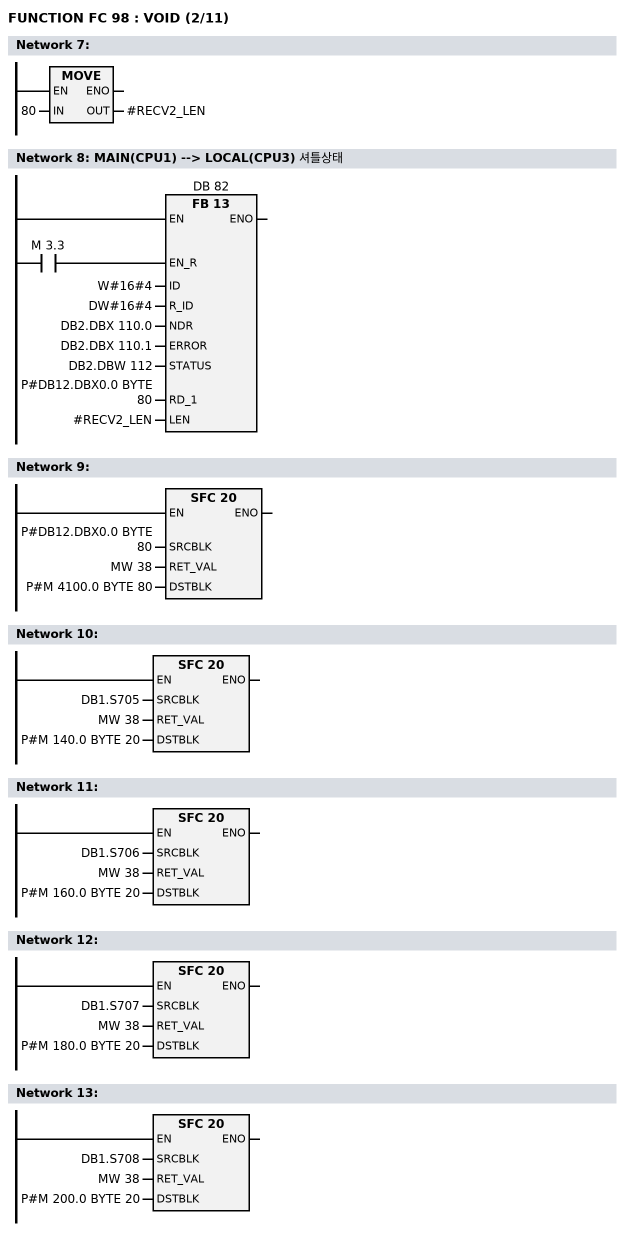

      L     80;
      T     #RECV2_LEN;
      NOP   0;
NETWORK
TITLE =MAIN(CPU1) --> LOCAL(CPU3) 셔틀상태

      A     M      3.3;
      =     L     22.0;
      BLD   103;
      CALL FB    13 , DB    82 (
           EN_R                     := L     22.0,
           ID                       := W#16#4,
           R_ID                     := DW#16#4,
           NDR                      := DB2.DBX  110.0,
           ERROR                    := DB2.DBX  110.1,
           STATUS                   := DB2.DBW  112,
           RD_1                     := P#DB12.DBX0.0 BYTE 80,
           LEN                      := #RECV2_LEN);
      NOP   0;
NETWORK
TITLE =

      CALL SFC   20 (
           SRCBLK                   := P#DB12.DBX0.0 BYTE 80,
           RET_VAL                  := MW    38,
           DSTBLK                   := P#M 4100.0 BYTE 80);
      NOP   0;
NETWORK
TITLE =

      CALL SFC   20 (
           SRCBLK                   := DB1.S705,
           RET_VAL                  := MW    38,
           DSTBLK                   := P#M 140.0 BYTE 20);
      NOP   0;
NETWORK
TITLE =

      CALL SFC   20 (
           SRCBLK                   := DB1.S706,
           RET_VAL                  := MW    38,
           DSTBLK                   := P#M 160.0 BYTE 20);
      NOP   0;
NETWORK
TITLE =

      CALL SFC   20 (
           SRCBLK                   := DB1.S707,
           RET_VAL                  := MW    38,
           DSTBLK                   := P#M 180.0 BYTE 20);
      NOP   0;
NETWORK
TITLE =

      CALL SFC   20 (
           SRCBLK                   := DB1.S708,
           RET_VAL                  := MW    38,
           DSTBLK                   := P#M 200.0 BYTE 20);
      NOP   0;
NETWORK
TITLE =
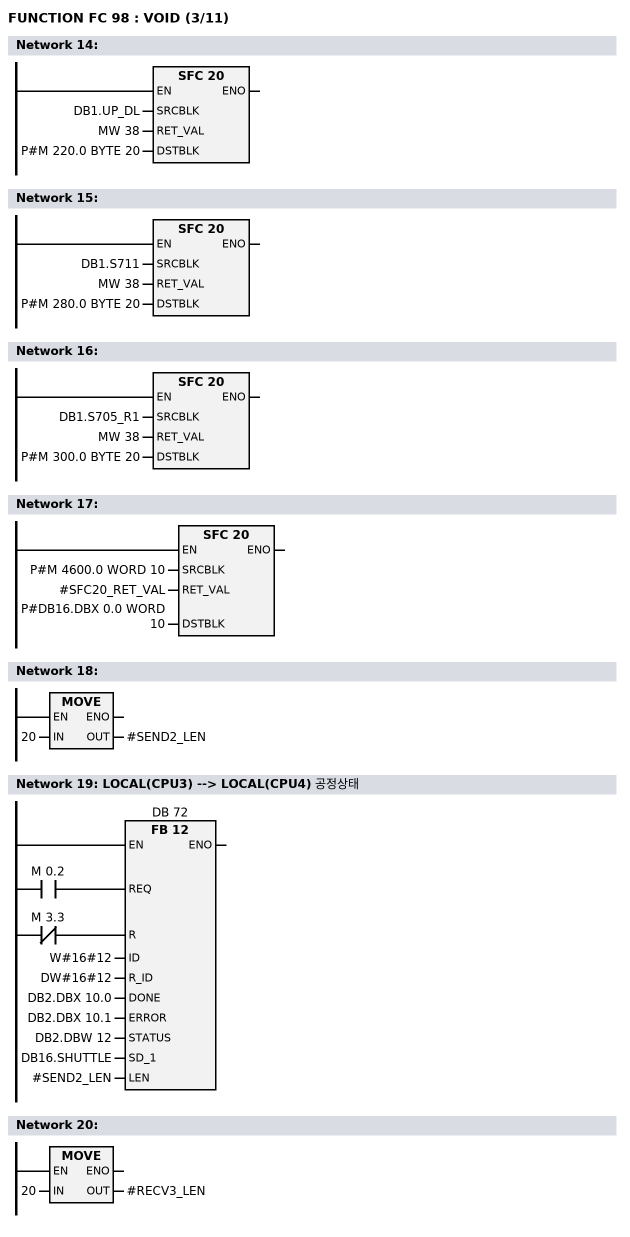

      CALL SFC   20 (
           SRCBLK                   := DB1.UP_DL,
           RET_VAL                  := MW    38,
           DSTBLK                   := P#M 220.0 BYTE 20);
      NOP   0;
NETWORK
TITLE =

      CALL SFC   20 (
           SRCBLK                   := DB1.S711,
           RET_VAL                  := MW    38,
           DSTBLK                   := P#M 280.0 BYTE 20);
      NOP   0;
NETWORK
TITLE =

      CALL SFC   20 (
           SRCBLK                   := DB1.S705_R1,
           RET_VAL                  := MW    38,
           DSTBLK                   := P#M 300.0 BYTE 20);
      NOP   0;
NETWORK
TITLE =

      CALL SFC   20 (
           SRCBLK                   := P#M 4600.0 WORD 10,
           RET_VAL                  := #SFC20_RET_VAL,
           DSTBLK                   := P#DB16.DBX 0.0 WORD 10);
      NOP   0;
NETWORK
TITLE =

      L     20;
      T     #SEND2_LEN;
      NOP   0;
NETWORK
TITLE =LOCAL(CPU3) --> LOCAL(CPU4) 공정상태

